           //"DI2"."SPARE1" := "BA010AZCRDI2.00";
           "DI2"."CONTROL POWER SMPS DC OK E6104PWS" := "BA010AZCRMP102.01";
           "DI2"."ET200MP I/O OUTPUT POWER TRIPPED E6154CB" := "BA010AZCRMP102.02";
           "DI2"."JUNCTION BOX CONTROL POWER TRIPPED E6180CB" := "BA010AZCRMP102.03";
           "DI2"."CLASS 2 SMPS POWER TRIPPED E6204CB" := "BA010AZCRMP102.04";
           "DI2"."CLASS 2 SMPS MONITORING E6206PWS" := "BA010AZCRMP102.05";
           "DI2"."ET200ECO PN-1 POWER TRIPPED E6220CB" := "BA010AZCRMP102.06";
           "DI2"."ET200ECO PN-2 POWER TRIPPED E6224CB" := "BA010AZCRMP102.07";
           "DI2"."ET200ECO PN-3 POWER TRIPPED E6228CB" := "BA010AZCRMP102.10";
           //"DI2"."SPARE2" := "BA010AZCRDI2.09";
           "DI2"."PANEL FAN POWER TRIPPED E6304CB" := "BA010AZCRMP102.12";
           //"DI2"."SPARE3" := "BA010AZCRDI2.11";
           "DI2"."CONTROLLER POWER SMPS DC OK E6404PWS" := "BA010AZCRMP102.14";
           "DI2"."CONTROLLER DC POWER TRIPPED E6406CB" := "BA010AZCRMP102.15";
           "DI2"."SERVO CONTROL POWER TRIPPED E6416CB" := "BA010AZCRMP102.16";
           "DI2"."MANIFOLD-1 CONTROL POWER TRIPPED E6422CB" := "BA010AZCRMP102.17";
           //"DI2"."SPARE4" := "BA010AZCRDI2.16";
           "DI2"."RFID POWER TRIPPED E6456CB" := "BA010AZCRMP102.21";
           "DI2"."QR READER POWER TRIPPED E6462CB" := "BA010AZCRMP102.22";
           "DI2"."QR READER POWER TRIPPED E6468CB" := "BA010AZCRMP102.23";
           //"DI2"."SPARE5" := "BA010AZCRDI2.20";
           //"DI2"."SPARE6" := "BA010AZCRDI2.21";
           "DI2"."CONTROLLER POWER SMPS DC OK E6704PWS" := "BA010AZCRMP102.26";
           "DI2"."CONTROLLER DC POWER TRIPPED E6706CB" := "BA010AZCRMP102.27";
           "DI2"."HANDY QR READER POWER TRIPPED E6716CB" := "BA010AZCRMP102.30";
           "DI2"."VISION CONTROLLER POWER TRIPPED E6722CB" := "BA010AZCRMP102.31";
           "DI2"."LINE LASER MODULE-1 POWER TRIPPED E6728CB" := "BA010AZCRMP102.32";
           "DI2"."LINE LASER MODULE-2 POWER TRIPPED E6734CB" := "BA010AZCRMP102.33";
           "DI2"."EPC CONTROLLER-1 POWER TRIPPED E6756CB" := "BA010AZCRMP102.34";
           "DI2"."EPC CONTROLLER-2 POWER TRIPPED E6762CB" := "BA010AZCRMP102.35";
           "DI2"."EPC CONTROLLER-3 POWER TRIPPED E6768CB" := "BA010AZCRMP102.36";
           "DI2"."DRIVE-CLIQ HUB POWER TRIPPED E6774CB" := "BA010AZCRMP102.37";


       END_REGION

       REGION DI3

           "DI3"."EQUIPMENT LED POWER TRIPPED E6780CB" := "BA010AZCRMP103.00";
           "DI3"."MOTOR POWER MC COIL POWER TRIPPED E6786CB" := "BA010AZCRMP103.01";
           "DI3"."SAFETY POWER SMPS DC OK E6804PWS" := "BA010AZCRMP103.02";
           "DI3"."SAFETY DC POWER TRIPPED E6808CB" := "BA010AZCRMP103.03";
           "DI3"."ET200SP I/O SAFETY POWER TRIPPED E6816CB" := "BA010AZCRMP103.04";
           "DI3"."JUNCTION BOX CONTROL POWER TRIPPED E6836CB" := "BA010AZCRMP103.05";
           "DI3"."ET200ECO PN-SAFETY-1 POWER TRIPPED E6856CB" := "BA010AZCRMP103.06";
           //"DI3"."SPARE1" := "BA010AZCRDI3.07";
           //"DI3"."SPARE2" := "BA010AZCRDI3.08";
           //"DI3"."SPARE3" := "BA010AZCRDI3.09";
           //"DI3"."SPARE4" := "BA010AZCRDI3.10";
           //"DI3"."SPARE5" := "BA010AZCRDI3.11";
           //"DI3"."SPARE6" := "BA010AZCRDI3.12";
           //"DI3"."SPARE7" := "BA010AZCRDI3.13";
           //"DI3"."SPARE8" := "BA010AZCRDI3.14";
           //"DI3"."SPARE9" := "BA010AZCRDI3.15";
           //"DI3"."SPARE10" := "BA010AZCRDI3.16";
           //"DI3"."SPARE11" := "BA010AZCRDI3.17";
           //"DI3"."SPARE12" := "BA010AZCRDI3.18";
           //"DI3"."SPARE13" := "BA010AZCRDI3.19";
           //"DI3"."SPARE14" := "BA010AZCRDI3.20";
           //"DI3"."SPARE15" := "BA010AZCRDI3.21";
           //"DI3"."SPARE16" := "BA010AZCRDI3.22";
           //"DI3"."SPARE17" := "BA010AZCRDI3.23";
           //"DI3"."SPARE18" := "BA010AZCRDI3.24";
           //"DI3"."SPARE19" := "BA010AZCRDI3.25";
           //"DI3"."SPARE20" := "BA010AZCRDI3.26";
           //"DI3"."SPARE21" := "BA010AZCRDI3.27";
           //"DI3"."SPARE22" := "BA010AZCRDI3.28";
           //"DI3"."SPARE23" := "BA010AZCRDI3.29";
           //"DI3"."SPARE24" := "BA010AZCRDI3.30";
           //"DI3"."SPARE25" := "BA010AZCRDI3.31";


       END_REGION

       REGION DQ1

           "DQ1"."EQUIPMENT LED LAMP RELAY ON" := "BA010AZCRMP104.00";
           //"DQ1"."SPARE1" := "BA010AZCRDQ1.01";
           //"DQ1"."SPARE2" := "BA010AZCRDQ1.02";
           "DQ1"."CLASS2 SMPS ALARM RESET" := "BA010AZCRMP104.03";
           //"DQ1"."SPARE3" := "BA010AZCRDQ1.04";
           //"DQ1"."SPARE4" := "BA010AZCRDQ1.05";
           //"DQ1"."SPARE5" := "BA010AZCRDQ1.06";
           //"DQ1"."SPARE6" := "BA010AZCRDQ1.07";
           //"DQ1"."SPARE7" := "BA010AZCRDQ1.08";
           //"DQ1"."SPARE8" := "BA010AZCRDQ1.09";
           //"DQ1"."SPARE9" := "BA010AZCRDQ1.10";
           //"DQ1"."SPARE10" := "BA010AZCRDQ1.11";
           //"DQ1"."SPARE11" := "BA010AZCRDQ1.12";
           //"DQ1"."SPARE12" := "BA010AZCRDQ1.13";
           //"DQ1"."SPARE13" := "BA010AZCRDQ1.14";
           //"DQ1"."SPARE14" := "BA010AZCRDQ1.15";
           //"DQ1"."SPARE15" := "BA010AZCRDQ1.16";
           //"DQ1"."SPARE16" := "BA010AZCRDQ1.17";
           //"DQ1"."SPARE17" := "BA010AZCRDQ1.18";
           //"DQ1"."SPARE18" := "BA010AZCRDQ1.19";
           //"DQ1"."SPARE19" := "BA010AZCRDQ1.20";
           //"DQ1"."SPARE20" := "BA010AZCRDQ1.21";
           //"DQ1"."SPARE21" := "BA010AZCRDQ1.22";
           //"DQ1"."SPARE22" := "BA010AZCRDQ1.23";
           //"DQ1"."SPARE23" := "BA010AZCRDQ1.24";
           //"DQ1"."SPARE24" := "BA010AZCRDQ1.25";
           //"DQ1"."SPARE25" := "BA010AZCRDQ1.26";
           //"DQ1"."SPARE26" := "BA010AZCRDQ1.27";
           //"DQ1"."SPARE27" := "BA010AZCRDQ1.28";
           //"DQ1"."SPARE28" := "BA010AZCRDQ1.29";
           //"DQ1"."SPARE29" := "BA010AZCRDQ1.30";
           //"DQ1"."SPARE30" := "BA010AZCRDQ1.31";


       END_REGION

       REGION FDI1

           "FDI1"."MANIFOLD-1 SOL POWER MC FEEDBACK" := "BA010AZCRMP105.00";
           "FDI1"."MANIFOLD-2 SOL POWER MC FEEDBACK" := "BA010AZCRMP105.01";
           //"FDI1"."SPARE1" := "BA010AZCRFDI1.02";
           //"FDI1"."SPARE2" := "BA010AZCRFDI1.03";
           "FDI1"."FFU POWER MC 1 FEEDBACK" := "BA010AZCRMP105.04";
           "FDI1"."FFU POWER MC 2 FEEDBACK" := "BA010AZCRMP105.05";
           //"FDI1"."SPARE3" := "BA010AZCRFDI1.06";
           //"FDI1"."SPARE4" := "BA010AZCRFDI1.07";


       END_REGION

       REGION FDQ1

           "FDQ1"."MANIFOLD-1 SOL POWER MC ON" := "BA010AZCRMP106.00";
           //"FDQ1"."SPARE1" := "BA010AZCRFDQ1.01";
           //"FDQ1"."SPARE2" := "BA010AZCRFDQ1.02";
           //"FDQ1"."SPARE3" := "BA010AZCRFDQ1.03";
           "FDQ1"."FFU POWER MC ON 1" := "BA010AZCRMP106.04";
           "FDQ1"."FFU POWER MC ON 2" := "BA010AZCRMP106.05";
           //"FDQ1"."SPARE4" := "BA010AZCRFDQ1.06";
           //"FDQ1"."SPARE5" := "BA010AZCRFDQ1.07";


       END_REGION


   END_REGION
END_FUNCTION

FUNCTION_BLOCK "CallInterfaceSignals"   // FB38, LAD
TITLE = CallInterfaceSignals
AUTHOR : SICAR
FAMILY : Diag
VERSION : 1.0
// Der Baustein dient als Aufrufschnittstelle für den Funktionsbaustein „LSicar_InterfaceSignalsBool“. Er ist als Funktionsbaustein ausgeführt, um die intern aufgerufenen FBs mittels Multiinstanzen realisieren zu können.  
// Die Funktionsbausteine und das zugehörige WinCC-Bild sind für 16 Signaldatensätze („Schnittstelle Signale 01“ … „Schnittstellen Signale 16“) mit jeweils 32 boolschen Signalen vorgesehen.  
// 
// **PLC-Datentypen**  
//  LSicar_typeInterfaceSignalsBool 
//  typeInterfaceSignalsHmi 
//  LSicar _typeInterfaceSignals 
// 
// **WinCC-Diagnosebild**  
// 
// ![Icon](_Icon/reference.PNG)
// 
// siehe ..\Library Types\LSicar_InterfaceSignalsBool.pdf  
// 
//  
// 
// **Beispielaufruf**  
// Abbildung in Kontaktplan (KOP).  D:\Software\Symbols_Icons\BMPs-JPGs-PNGs\Verschiedene\symb_user_goto_transparent.pngEin lauffähiger Programm-Aufruf hierzu ist im „SICAR-StartUp“-Projekt enthalten.  
// 
// **Aufrufschnittstelle**  
// Der Baustein wird einmalig im zyklischen Programm aufgerufen.  
// 
// **Intern verwendete „Erweiterte Anweisungen / Bausteine“**  
// ..\Library Types\LSicar_InterfaceSignalsBool.pdf
// The block serves as a calling interface of the block “InterfaceSignalsBool“. The block is designed as function block in order to implement the block calls as multi-instances.
// stored: IsIECCheckEnabled true, MemoryReserve 100, SetENOAutomatically true
   VAR
      statReadValueHmi : Bool;   // HMI: Lese Signalwert / HMI: Read value signal
      statSelectSignalsHmi : USInt := 1;   // HMI: Angewählte Interface Schnittstelle (1..16) / HMI: Selected interface signals (1..16)
      statSelectSignalsOld { ExternalAccessible := 'False'; ExternalVisible := 'False'; ExternalWritable := 'False'} : USInt;   // Altwert: Angewählte Interface Schnittstelle / Old value: Selected interface signals
      statRisEdgeReadName { ExternalAccessible := 'False'; ExternalVisible := 'False'; ExternalWritable := 'False'} : Bool;   // Steigende Flanke / Rising edge
      statPosPulseReadName : Bool;   // Positiver Impuls / Positive pulse
   END_VAR
   VAR RETAIN
      statInterfaceSignalsHmi : Array[0..70] of "typeInterfaceSignalsHmi";   // HMI: Beschreibung, Wert und Symbolischer Name / HMI: Description, value and symbolic name
   END_VAR
   VAR
      instSignalsLeft { ExternalAccessible := 'False'; ExternalVisible := 'False'; ExternalWritable := 'False'} : Array[0..70] of "LAF_InterfaceSignalsBool";   // Schnittstellen Signale Bild 1 links / interface signals screen left
      instSignalsRight { ExternalAccessible := 'False'; ExternalVisible := 'False'; ExternalWritable := 'False'} : Array[0..70] of "LAF_InterfaceSignalsBool";   // Schnittstellen Signale Bild 1 rechts / interface signals screen right
   END_VAR
   VAR_TEMP
      tempLoopCounter : DInt;   // temp. Schleifenzähler / temp. Loop Counter
   END_VAR
   VAR_TEMP   // added for the SCL form of the ladder/FBD networks
      _w1 : Bool;
   END_VAR
BEGIN

REGION Network 1: Beschreibung / BLOCK INFO HEADER
   // **Betriebsart Automatik / Hand**  
   // Der Baustein ist keiner Betriebsart / Betriebsartenbereich zugeordnet.  
   // 
   // **Alarme**  
   // Der Baustein generiert keine Alarme.  
   // 
   // #### PLC-Datentypen  
   // Verwendete PLC-Datentypen für den SPS-Programmbaustein und das zugehörige WinCC-Bild.  
   // 
   // {.pageWidth}
   // ![Image](CallInterfaceSignals/de/image1.PNG)
   //  
   //  
   // #### Bausteinaufrufe 
   // Der Baustein “LSicar_InterfaceSignalsBool“ wird in diesem FB als Multi-Instanz aufgerufen, entspr. nebenstehender beispielhafter Darstellung.  
   // 
   // {.pageWidth}
   // ![Image](CallInterfaceSignals/de/image2.PNG)
   //  
   // Um einen neuen FB aufzurufen, ziehen Sie den FB in ein neues Netzwerk, wählen Sie „Multiinstanz“ aus, vergeben Sie einen Namen und parametrieren Sie den FB-Aufruf.  
   // 
   // {.pageWidth}
   // ![Image](CallInterfaceSignals/de/image3.PNG)
   //  
   //  
   // #### Weitere Hinweise 
   // 
   // #### Updateinfo 
   // 
   // #### Weitere Dokumente 
   // 
   // ![Icon](_Icon/reference.PNG)
   // 
   // ..\Library Types\LSicar_InterfaceSignalsBool.pdf
   // SIEMENS AG / (c)Copyright 2023
   // ------------------------------------------------------------------------------
   // Title:            CallInterfaceSignals (FB38)
   // Comment/Function: The block serves as a calling interface of the block “InterfaceSignalsBool“. The block is designed as function block in order to implement the block calls as multi-instances. 
   // Library/Family:   Diag
   // Author:           SICAR
   // Tested with:      ---
   // Engineering:      TIA Portal V19
   // Restrictions:     -
   // Requirements:     ---
   // ------------------------------------------------------------------------------
   // Change log table:
   // Version  | Date       | Expert in charge       | Changes applied
   // ---------|------------|------------------------|------------------------------
   // 01.00.00 | 11.12.2023 | SICAR
   //                         First released version
END_REGION

REGION Network 2: DESCRIPTION
   // Function block and corresponding WinCC screen are prepared for 16 data sets (“InterfaceSignals01“ through .”InterfaceSignals16“) with 32 Boolean signals each.  
   // 
   // **PLC-Data types**   
   // 
   // * LSicar_typeInterfaceSignalsBool 
   // * LSicar _typeInterfaceSignals 
   // * typeInterfaceSignalsHmi 
   // 
   // **WinCC-Faceplate**  
   // 
   // <None> 
   // 
   // **WinCC Diagnostic screen**   
   // 
   // See: ..\Library Types\LSicar_InterfaceSignalsBool.pdf  
   // 
   // **Block call example** 
   // 
   // View in ladder-logic (LAD), without parameter settings.  
   // An executable program call is available in the “SICAR-Startup” project.  
   // 
   // **Calling interface**  
   // 
   // The block is be called once in the cyclic program.  
   // 
   // **Internally used „Extended instructions / blocks“**  
   // 
   // See: ..\Library Types\LSicar_InterfaceSignalsBool.pdf
END_REGION

REGION Network 3: Initialisierung Loop_1 / Initialization Loop_1
   // Vorbesetzen des Schleifenindex / Preset the loop index
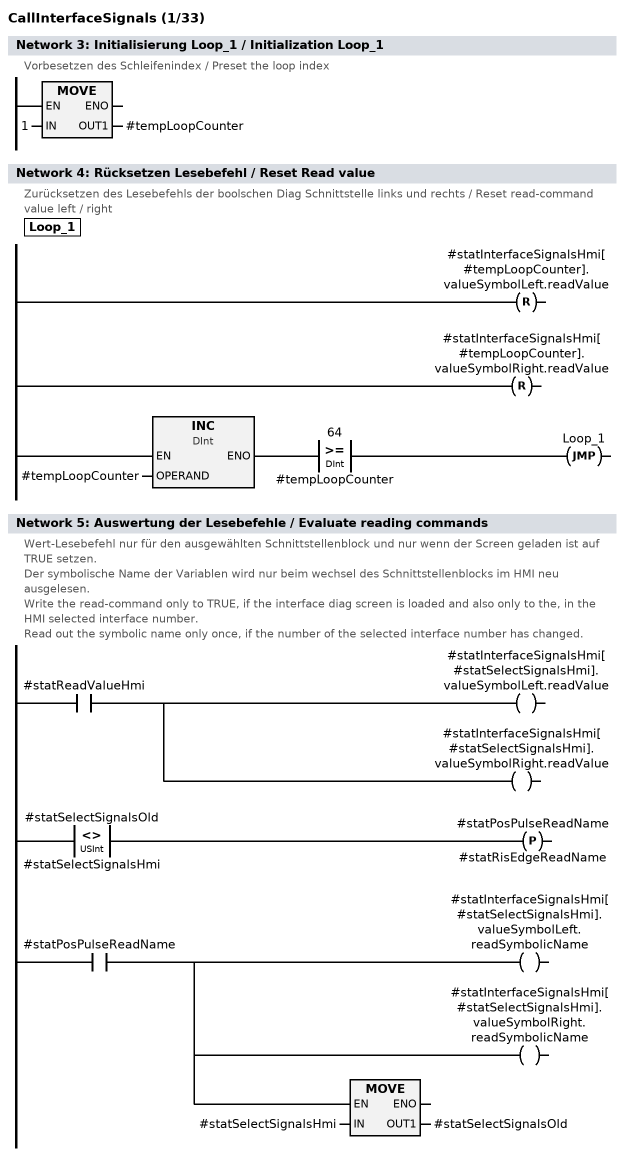
   RUNG wire#powerrail
      Move(in := 1, out1 => #tempLoopCounter)
   END_RUNG
   // the same network as SCL:
   #tempLoopCounter := 1;
END_REGION

REGION Network 4: Rücksetzen Lesebefehl / Reset Read value
   // Zurücksetzen des Lesebefehls der boolschen Diag Schnittstelle links und rechts / Reset read-command value left / right
   Label( Loop_1 )
   RUNG wire#powerrail
      R_Coil( #statInterfaceSignalsHmi[#tempLoopCounter].valueSymbolLeft.readValue )
   END_RUNG
   RUNG wire#powerrail
      R_Coil( #statInterfaceSignalsHmi[#tempLoopCounter].valueSymbolRight.readValue )
   END_RUNG
   RUNG wire#powerrail
      { S7_Templates := "DestType := DInt" } Inc( #tempLoopCounter )
      { S7_Templates := "SrcType := DInt" } GE_Contact(in1 := 64, in2 := #tempLoopCounter)
      JumpCoil( Loop_1 )
   END_RUNG
   // the same network as SCL:
   Loop_1:
   #statInterfaceSignalsHmi[#tempLoopCounter].valueSymbolLeft.readValue := FALSE;
   #statInterfaceSignalsHmi[#tempLoopCounter].valueSymbolRight.readValue := FALSE;
   #tempLoopCounter := #tempLoopCounter + 1;
   IF 64 >= #tempLoopCounter THEN GOTO Loop_1; END_IF;
END_REGION

REGION Network 5: Auswertung der Lesebefehle / Evaluate reading commands
   // Wert-Lesebefehl nur für den ausgewählten Schnittstellenblock und nur wenn der Screen geladen ist auf TRUE setzen.
   // Der symbolische Name der Variablen wird nur beim wechsel des Schnittstellenblocks im HMI neu ausgelesen.
   // Write the read-command only to TRUE, if the interface diag screen is loaded and also only to the, in the HMI selected interface number.
   // Read out the symbolic name only once, if the number of the selected interface number has changed.
   #statInterfaceSignalsHmi[#statSelectSignalsHmi].valueSymbolLeft.readValue := #statReadValueHmi;
   #statInterfaceSignalsHmi[#statSelectSignalsHmi].valueSymbolRight.readValue := #statReadValueHmi;
   #_w1 := #statSelectSignalsOld <> #statSelectSignalsHmi;
   #statPosPulseReadName := #_w1 AND NOT #statRisEdgeReadName;   // rising edge
   #statRisEdgeReadName := #_w1;
   #statInterfaceSignalsHmi[#statSelectSignalsHmi].valueSymbolLeft.readSymbolicName := #statPosPulseReadName;
   #statInterfaceSignalsHmi[#statSelectSignalsHmi].valueSymbolRight.readSymbolicName := #statPosPulseReadName;
   IF #statPosPulseReadName THEN #statSelectSignalsOld := #statSelectSignalsHmi; END_IF;
END_REGION

REGION Network 6: Interface Signals 01 -Example: Model PosDev+Lifter - IN/OUT- / Interface Signals Stack30
   // Aufruf des Schnittstellen Signal Bausteins Ba-Bereich 1 / Call the interface signals bool blocks of system tags
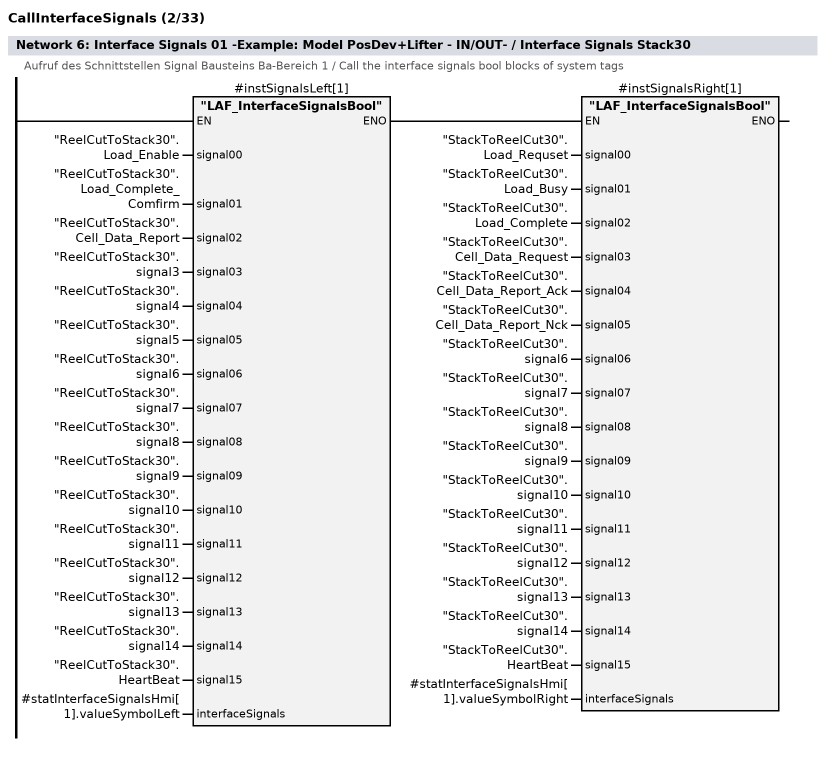
   RUNG wire#powerrail
      #instSignalsLeft[1](signal00 := "ReelCutToStack30".Load_Enable, signal01 := "ReelCutToStack30".Load_Complete_Comfirm, signal02 := "ReelCutToStack30".Cell_Data_Report, signal03 := "ReelCutToStack30".signal3, signal04 := "ReelCutToStack30".signal4, signal05 := "ReelCutToStack30".signal5, signal06 := "ReelCutToStack30".signal6, signal07 := "ReelCutToStack30".signal7, signal08 := "ReelCutToStack30".signal8, signal09 := "ReelCutToStack30".signal9, signal10 := "ReelCutToStack30".signal10, signal11 := "ReelCutToStack30".signal11, signal12 := "ReelCutToStack30".signal12, signal13 := "ReelCutToStack30".signal13, signal14 := "ReelCutToStack30".signal14, signal15 := "ReelCutToStack30".HeartBeat, interfaceSignals := #statInterfaceSignalsHmi[1].valueSymbolLeft)
      #instSignalsRight[1](signal00 := "StackToReelCut30".Load_Requset, signal01 := "StackToReelCut30".Load_Busy, signal02 := "StackToReelCut30".Load_Complete, signal03 := "StackToReelCut30".Cell_Data_Request, signal04 := "StackToReelCut30".Cell_Data_Report_Ack, signal05 := "StackToReelCut30".Cell_Data_Report_Nck, signal06 := "StackToReelCut30".signal6, signal07 := "StackToReelCut30".signal7, signal08 := "StackToReelCut30".signal8, signal09 := "StackToReelCut30".signal9, signal10 := "StackToReelCut30".signal10, signal11 := "StackToReelCut30".signal11, signal12 := "StackToReelCut30".signal12, signal13 := "StackToReelCut30".signal13, signal14 := "StackToReelCut30".signal14, signal15 := "StackToReelCut30".HeartBeat, interfaceSignals := #statInterfaceSignalsHmi[1].valueSymbolRight)
   END_RUNG
   // the same network as SCL:
   #instSignalsLeft[1](signal00 := "ReelCutToStack30".Load_Enable,   // "LAF_InterfaceSignalsBool"
                       signal01 := "ReelCutToStack30".Load_Complete_Comfirm,
                       signal02 := "ReelCutToStack30".Cell_Data_Report,
                       signal03 := "ReelCutToStack30".signal3,
                       signal04 := "ReelCutToStack30".signal4,
                       signal05 := "ReelCutToStack30".signal5,
                       signal06 := "ReelCutToStack30".signal6,
                       signal07 := "ReelCutToStack30".signal7,
                       signal08 := "ReelCutToStack30".signal8,
                       signal09 := "ReelCutToStack30".signal9,
                       signal10 := "ReelCutToStack30".signal10,
                       signal11 := "ReelCutToStack30".signal11,
                       signal12 := "ReelCutToStack30".signal12,
                       signal13 := "ReelCutToStack30".signal13,
                       signal14 := "ReelCutToStack30".signal14,
                       signal15 := "ReelCutToStack30".HeartBeat,
                       interfaceSignals := #statInterfaceSignalsHmi[1].valueSymbolLeft,
                       ENO => #_w1);
   IF #_w1 THEN
       #instSignalsRight[1](signal00 := "StackToReelCut30".Load_Requset,   // "LAF_InterfaceSignalsBool"
                            signal01 := "StackToReelCut30".Load_Busy,
                            signal02 := "StackToReelCut30".Load_Complete,
                            signal03 := "StackToReelCut30".Cell_Data_Request,
                            signal04 := "StackToReelCut30".Cell_Data_Report_Ack,
                            signal05 := "StackToReelCut30".Cell_Data_Report_Nck,
                            signal06 := "StackToReelCut30".signal6,
                            signal07 := "StackToReelCut30".signal7,
                            signal08 := "StackToReelCut30".signal8,
                            signal09 := "StackToReelCut30".signal9,
                            signal10 := "StackToReelCut30".signal10,
                            signal11 := "StackToReelCut30".signal11,
                            signal12 := "StackToReelCut30".signal12,
                            signal13 := "StackToReelCut30".signal13,
                            signal14 := "StackToReelCut30".signal14,
                            signal15 := "StackToReelCut30".HeartBeat,
                            interfaceSignals := #statInterfaceSignalsHmi[1].valueSymbolRight);
   END_IF;
END_REGION

REGION Network 7: Interface Signals 01 -Example: Model PosDev+Lifter - IN/OUT- / Interface Signals Stack40
   // Aufruf des Schnittstellen Signal Bausteins Ba-Bereich 1 / Call the interface signals bool blocks of system tags
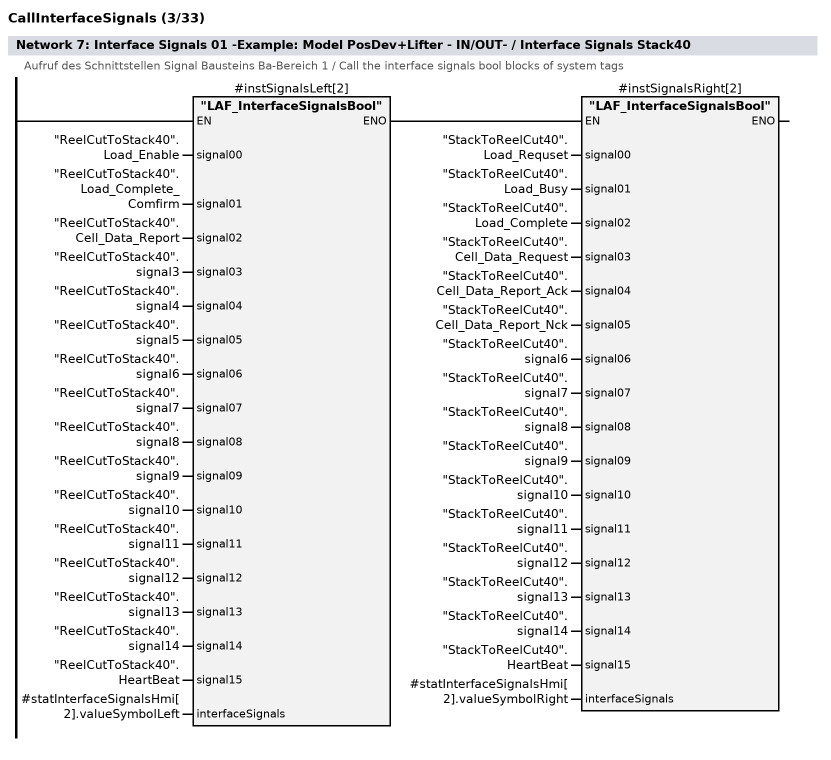
   RUNG wire#powerrail
      #instSignalsLeft[2](signal00 := "ReelCutToStack40".Load_Enable, signal01 := "ReelCutToStack40".Load_Complete_Comfirm, signal02 := "ReelCutToStack40".Cell_Data_Report, signal03 := "ReelCutToStack40".signal3, signal04 := "ReelCutToStack40".signal4, signal05 := "ReelCutToStack40".signal5, signal06 := "ReelCutToStack40".signal6, signal07 := "ReelCutToStack40".signal7, signal08 := "ReelCutToStack40".signal8, signal09 := "ReelCutToStack40".signal9, signal10 := "ReelCutToStack40".signal10, signal11 := "ReelCutToStack40".signal11, signal12 := "ReelCutToStack40".signal12, signal13 := "ReelCutToStack40".signal13, signal14 := "ReelCutToStack40".signal14, signal15 := "ReelCutToStack40".HeartBeat, interfaceSignals := #statInterfaceSignalsHmi[2].valueSymbolLeft)
      #instSignalsRight[2](signal00 := "StackToReelCut40".Load_Requset, signal01 := "StackToReelCut40".Load_Busy, signal02 := "StackToReelCut40".Load_Complete, signal03 := "StackToReelCut40".Cell_Data_Request, signal04 := "StackToReelCut40".Cell_Data_Report_Ack, signal05 := "StackToReelCut40".Cell_Data_Report_Nck, signal06 := "StackToReelCut40".signal6, signal07 := "StackToReelCut40".signal7, signal08 := "StackToReelCut40".signal8, signal09 := "StackToReelCut40".signal9, signal10 := "StackToReelCut40".signal10, signal11 := "StackToReelCut40".signal11, signal12 := "StackToReelCut40".signal12, signal13 := "StackToReelCut40".signal13, signal14 := "StackToReelCut40".signal14, signal15 := "StackToReelCut40".HeartBeat, interfaceSignals := #statInterfaceSignalsHmi[2].valueSymbolRight)
   END_RUNG
   // the same network as SCL:
   #instSignalsLeft[2](signal00 := "ReelCutToStack40".Load_Enable,   // "LAF_InterfaceSignalsBool"
                       signal01 := "ReelCutToStack40".Load_Complete_Comfirm,
                       signal02 := "ReelCutToStack40".Cell_Data_Report,
                       signal03 := "ReelCutToStack40".signal3,
                       signal04 := "ReelCutToStack40".signal4,
                       signal05 := "ReelCutToStack40".signal5,
                       signal06 := "ReelCutToStack40".signal6,
                       signal07 := "ReelCutToStack40".signal7,
                       signal08 := "ReelCutToStack40".signal8,
                       signal09 := "ReelCutToStack40".signal9,
                       signal10 := "ReelCutToStack40".signal10,
                       signal11 := "ReelCutToStack40".signal11,
                       signal12 := "ReelCutToStack40".signal12,
                       signal13 := "ReelCutToStack40".signal13,
                       signal14 := "ReelCutToStack40".signal14,
                       signal15 := "ReelCutToStack40".HeartBeat,
                       interfaceSignals := #statInterfaceSignalsHmi[2].valueSymbolLeft,
                       ENO => #_w1);
   IF #_w1 THEN
       #instSignalsRight[2](signal00 := "StackToReelCut40".Load_Requset,   // "LAF_InterfaceSignalsBool"
                            signal01 := "StackToReelCut40".Load_Busy,
                            signal02 := "StackToReelCut40".Load_Complete,
                            signal03 := "StackToReelCut40".Cell_Data_Request,
                            signal04 := "StackToReelCut40".Cell_Data_Report_Ack,
                            signal05 := "StackToReelCut40".Cell_Data_Report_Nck,
                            signal06 := "StackToReelCut40".signal6,
                            signal07 := "StackToReelCut40".signal7,
                            signal08 := "StackToReelCut40".signal8,
                            signal09 := "StackToReelCut40".signal9,
                            signal10 := "StackToReelCut40".signal10,
                            signal11 := "StackToReelCut40".signal11,
                            signal12 := "StackToReelCut40".signal12,
                            signal13 := "StackToReelCut40".signal13,
                            signal14 := "StackToReelCut40".signal14,
                            signal15 := "StackToReelCut40".HeartBeat,
                            interfaceSignals := #statInterfaceSignalsHmi[2].valueSymbolRight);
   END_IF;
END_REGION

REGION Network 8: Interface Signals 01 -Example: Rack-ET200SP Standard IN/OUT- / Interface Signals Bk01
   // Aufruf des Schnittstellen Signal Bausteins Ba-Bereich 1 / Call the interface signals bool blocks of system tags
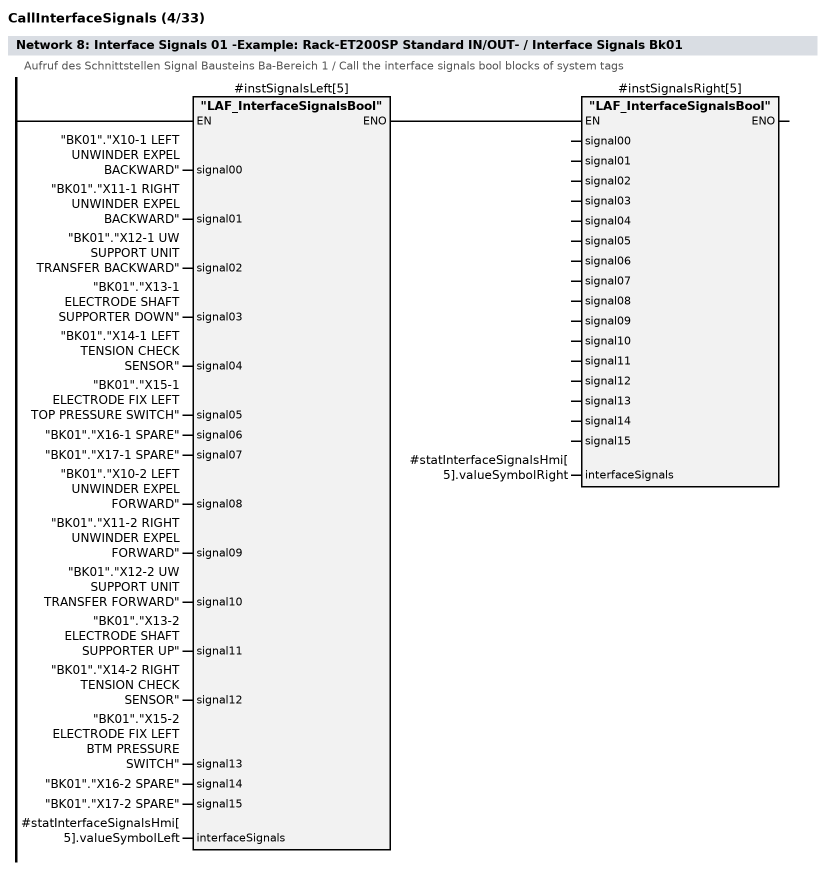
   RUNG wire#powerrail
      #instSignalsLeft[5](signal00 := "BK01"."X10-1 LEFT UNWINDER EXPEL BACKWARD", signal01 := "BK01"."X11-1 RIGHT UNWINDER EXPEL BACKWARD", signal02 := "BK01"."X12-1 UW SUPPORT UNIT TRANSFER BACKWARD", signal03 := "BK01"."X13-1 ELECTRODE SHAFT SUPPORTER DOWN", signal04 := "BK01"."X14-1 LEFT TENSION CHECK SENSOR", signal05 := "BK01"."X15-1 ELECTRODE FIX LEFT TOP PRESSURE SWITCH", signal06 := "BK01"."X16-1 SPARE", signal07 := "BK01"."X17-1 SPARE", signal08 := "BK01"."X10-2 LEFT UNWINDER EXPEL FORWARD", signal09 := "BK01"."X11-2 RIGHT UNWINDER EXPEL FORWARD", signal10 := "BK01"."X12-2 UW SUPPORT UNIT TRANSFER FORWARD", signal11 := "BK01"."X13-2 ELECTRODE SHAFT SUPPORTER UP", signal12 := "BK01"."X14-2 RIGHT TENSION CHECK SENSOR", signal13 := "BK01"."X15-2 ELECTRODE FIX LEFT BTM PRESSURE SWITCH", signal14 := "BK01"."X16-2 SPARE", signal15 := "BK01"."X17-2 SPARE", interfaceSignals := #statInterfaceSignalsHmi[5].valueSymbolLeft)
      #instSignalsRight[5](signal00 :=, signal01 :=, signal02 :=, signal03 :=, signal04 :=, signal05 :=, signal06 :=, signal07 :=, signal08 :=, signal09 :=, signal10 :=, signal11 :=, signal12 :=, signal13 :=, signal14 :=, signal15 :=, interfaceSignals := #statInterfaceSignalsHmi[5].valueSymbolRight)
   END_RUNG
   // the same network as SCL:
   #instSignalsLeft[5](signal00 := "BK01"."X10-1 LEFT UNWINDER EXPEL BACKWARD",   // "LAF_InterfaceSignalsBool"
                       signal01 := "BK01"."X11-1 RIGHT UNWINDER EXPEL BACKWARD",
                       signal02 := "BK01"."X12-1 UW SUPPORT UNIT TRANSFER BACKWARD",
                       signal03 := "BK01"."X13-1 ELECTRODE SHAFT SUPPORTER DOWN",
                       signal04 := "BK01"."X14-1 LEFT TENSION CHECK SENSOR",
                       signal05 := "BK01"."X15-1 ELECTRODE FIX LEFT TOP PRESSURE SWITCH",
                       signal06 := "BK01"."X16-1 SPARE",
                       signal07 := "BK01"."X17-1 SPARE",
                       signal08 := "BK01"."X10-2 LEFT UNWINDER EXPEL FORWARD",
                       signal09 := "BK01"."X11-2 RIGHT UNWINDER EXPEL FORWARD",
                       signal10 := "BK01"."X12-2 UW SUPPORT UNIT TRANSFER FORWARD",
                       signal11 := "BK01"."X13-2 ELECTRODE SHAFT SUPPORTER UP",
                       signal12 := "BK01"."X14-2 RIGHT TENSION CHECK SENSOR",
                       signal13 := "BK01"."X15-2 ELECTRODE FIX LEFT BTM PRESSURE SWITCH",
                       signal14 := "BK01"."X16-2 SPARE",
                       signal15 := "BK01"."X17-2 SPARE",
                       interfaceSignals := #statInterfaceSignalsHmi[5].valueSymbolLeft,
                       ENO => #_w1);
   IF #_w1 THEN
       #instSignalsRight[5](interfaceSignals := #statInterfaceSignalsHmi[5].valueSymbolRight);   // "LAF_InterfaceSignalsBool"
   END_IF;
END_REGION

REGION Network 9: Interface Signals Bk02
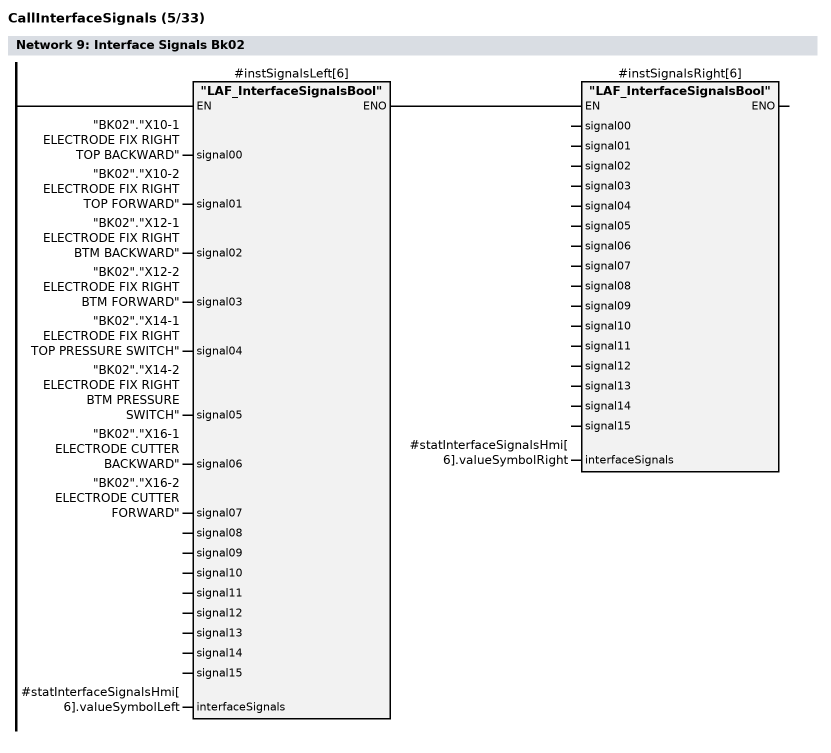
   RUNG wire#powerrail
      #instSignalsLeft[6](signal00 := "BK02"."X10-1 ELECTRODE FIX RIGHT TOP BACKWARD", signal01 := "BK02"."X10-2 ELECTRODE FIX RIGHT TOP FORWARD", signal02 := "BK02"."X12-1 ELECTRODE FIX RIGHT BTM BACKWARD", signal03 := "BK02"."X12-2 ELECTRODE FIX RIGHT BTM FORWARD", signal04 := "BK02"."X14-1 ELECTRODE FIX RIGHT TOP PRESSURE SWITCH", signal05 := "BK02"."X14-2 ELECTRODE FIX RIGHT BTM PRESSURE SWITCH", signal06 := "BK02"."X16-1 ELECTRODE CUTTER BACKWARD", signal07 := "BK02"."X16-2 ELECTRODE CUTTER FORWARD", signal08 :=, signal09 :=, signal10 :=, signal11 :=, signal12 :=, signal13 :=, signal14 :=, signal15 :=, interfaceSignals := #statInterfaceSignalsHmi[6].valueSymbolLeft)
      #instSignalsRight[6](signal00 :=, signal01 :=, signal02 :=, signal03 :=, signal04 :=, signal05 :=, signal06 :=, signal07 :=, signal08 :=, signal09 :=, signal10 :=, signal11 :=, signal12 :=, signal13 :=, signal14 :=, signal15 :=, interfaceSignals := #statInterfaceSignalsHmi[6].valueSymbolRight)
   END_RUNG
   // the same network as SCL:
   #instSignalsLeft[6](signal00 := "BK02"."X10-1 ELECTRODE FIX RIGHT TOP BACKWARD",   // "LAF_InterfaceSignalsBool"
                       signal01 := "BK02"."X10-2 ELECTRODE FIX RIGHT TOP FORWARD",
                       signal02 := "BK02"."X12-1 ELECTRODE FIX RIGHT BTM BACKWARD",
                       signal03 := "BK02"."X12-2 ELECTRODE FIX RIGHT BTM FORWARD",
                       signal04 := "BK02"."X14-1 ELECTRODE FIX RIGHT TOP PRESSURE SWITCH",
                       signal05 := "BK02"."X14-2 ELECTRODE FIX RIGHT BTM PRESSURE SWITCH",
                       signal06 := "BK02"."X16-1 ELECTRODE CUTTER BACKWARD",
                       signal07 := "BK02"."X16-2 ELECTRODE CUTTER FORWARD",
                       interfaceSignals := #statInterfaceSignalsHmi[6].valueSymbolLeft,
                       ENO => #_w1);
   IF #_w1 THEN
       #instSignalsRight[6](interfaceSignals := #statInterfaceSignalsHmi[6].valueSymbolRight);   // "LAF_InterfaceSignalsBool"
   END_IF;
END_REGION

REGION Network 10: Interface Signals 03 -Example: System flags & Clock flags- / Interface Signals Bk03
   // Aufruf des Schnittstellen Signal Bausteins für die Systemvariablen / Call the interface signals bool blocks of system tags
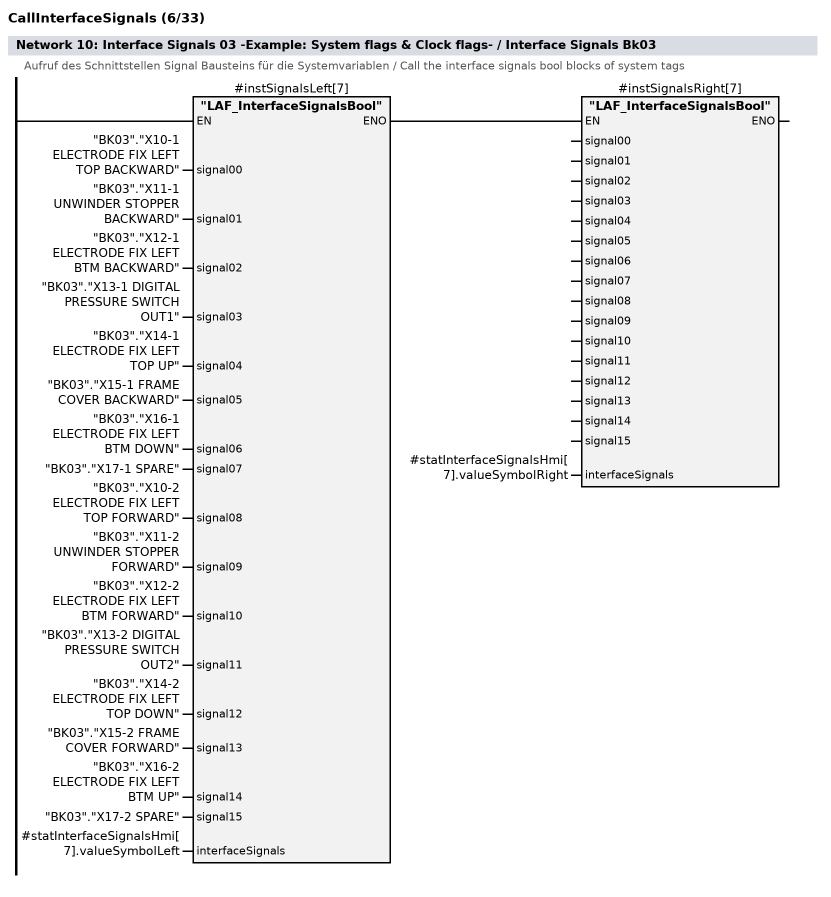
   RUNG wire#powerrail
      #instSignalsLeft[7](signal00 := "BK03"."X10-1 ELECTRODE FIX LEFT TOP BACKWARD", signal01 := "BK03"."X11-1 UNWINDER STOPPER BACKWARD", signal02 := "BK03"."X12-1 ELECTRODE FIX LEFT BTM BACKWARD", signal03 := "BK03"."X13-1 DIGITAL PRESSURE SWITCH OUT1", signal04 := "BK03"."X14-1 ELECTRODE FIX LEFT TOP UP", signal05 := "BK03"."X15-1 FRAME COVER BACKWARD", signal06 := "BK03"."X16-1 ELECTRODE FIX LEFT BTM DOWN", signal07 := "BK03"."X17-1 SPARE", signal08 := "BK03"."X10-2 ELECTRODE FIX LEFT TOP FORWARD", signal09 := "BK03"."X11-2 UNWINDER STOPPER FORWARD", signal10 := "BK03"."X12-2 ELECTRODE FIX LEFT BTM FORWARD", signal11 := "BK03"."X13-2 DIGITAL PRESSURE SWITCH OUT2", signal12 := "BK03"."X14-2 ELECTRODE FIX LEFT TOP DOWN", signal13 := "BK03"."X15-2 FRAME COVER FORWARD", signal14 := "BK03"."X16-2 ELECTRODE FIX LEFT BTM UP", signal15 := "BK03"."X17-2 SPARE", interfaceSignals := #statInterfaceSignalsHmi[7].valueSymbolLeft)
      #instSignalsRight[7](signal00 :=, signal01 :=, signal02 :=, signal03 :=, signal04 :=, signal05 :=, signal06 :=, signal07 :=, signal08 :=, signal09 :=, signal10 :=, signal11 :=, signal12 :=, signal13 :=, signal14 :=, signal15 :=, interfaceSignals := #statInterfaceSignalsHmi[7].valueSymbolRight)
   END_RUNG
   // the same network as SCL:
   #instSignalsLeft[7](signal00 := "BK03"."X10-1 ELECTRODE FIX LEFT TOP BACKWARD",   // "LAF_InterfaceSignalsBool"
                       signal01 := "BK03"."X11-1 UNWINDER STOPPER BACKWARD",
                       signal02 := "BK03"."X12-1 ELECTRODE FIX LEFT BTM BACKWARD",
                       signal03 := "BK03"."X13-1 DIGITAL PRESSURE SWITCH OUT1",
                       signal04 := "BK03"."X14-1 ELECTRODE FIX LEFT TOP UP",
                       signal05 := "BK03"."X15-1 FRAME COVER BACKWARD",
                       signal06 := "BK03"."X16-1 ELECTRODE FIX LEFT BTM DOWN",
                       signal07 := "BK03"."X17-1 SPARE",
                       signal08 := "BK03"."X10-2 ELECTRODE FIX LEFT TOP FORWARD",
                       signal09 := "BK03"."X11-2 UNWINDER STOPPER FORWARD",
                       signal10 := "BK03"."X12-2 ELECTRODE FIX LEFT BTM FORWARD",
                       signal11 := "BK03"."X13-2 DIGITAL PRESSURE SWITCH OUT2",
                       signal12 := "BK03"."X14-2 ELECTRODE FIX LEFT TOP DOWN",
                       signal13 := "BK03"."X15-2 FRAME COVER FORWARD",
                       signal14 := "BK03"."X16-2 ELECTRODE FIX LEFT BTM UP",
                       signal15 := "BK03"."X17-2 SPARE",
                       interfaceSignals := #statInterfaceSignalsHmi[7].valueSymbolLeft,
                       ENO => #_w1);
   IF #_w1 THEN
       #instSignalsRight[7](interfaceSignals := #statInterfaceSignalsHmi[7].valueSymbolRight);   // "LAF_InterfaceSignalsBool"
   END_IF;
END_REGION

REGION Network 11: Interface Signals 03 -Example: System flags & Clock flags- / Interface Signals Bk04
   // Aufruf des Schnittstellen Signal Bausteins für die Systemvariablen / Call the interface signals bool blocks of system tags
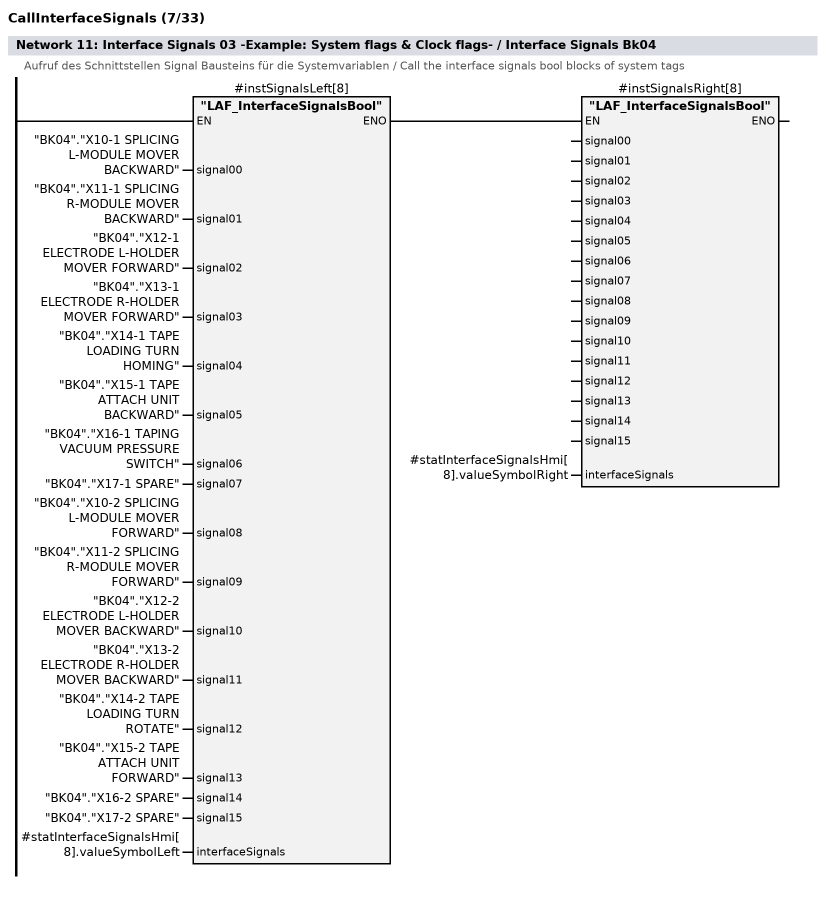
   RUNG wire#powerrail
      #instSignalsLeft[8](signal00 := "BK04"."X10-1 SPLICING L-MODULE MOVER BACKWARD", signal01 := "BK04"."X11-1 SPLICING R-MODULE MOVER BACKWARD", signal02 := "BK04"."X12-1 ELECTRODE L-HOLDER MOVER FORWARD", signal03 := "BK04"."X13-1 ELECTRODE R-HOLDER MOVER FORWARD", signal04 := "BK04"."X14-1 TAPE LOADING TURN HOMING", signal05 := "BK04"."X15-1 TAPE ATTACH UNIT BACKWARD", signal06 := "BK04"."X16-1 TAPING VACUUM PRESSURE SWITCH", signal07 := "BK04"."X17-1 SPARE", signal08 := "BK04"."X10-2 SPLICING L-MODULE MOVER FORWARD", signal09 := "BK04"."X11-2 SPLICING R-MODULE MOVER FORWARD", signal10 := "BK04"."X12-2 ELECTRODE L-HOLDER MOVER BACKWARD", signal11 := "BK04"."X13-2 ELECTRODE R-HOLDER MOVER BACKWARD", signal12 := "BK04"."X14-2 TAPE LOADING TURN ROTATE", signal13 := "BK04"."X15-2 TAPE ATTACH UNIT FORWARD", signal14 := "BK04"."X16-2 SPARE", signal15 := "BK04"."X17-2 SPARE", interfaceSignals := #statInterfaceSignalsHmi[8].valueSymbolLeft)
      #instSignalsRight[8](signal00 :=, signal01 :=, signal02 :=, signal03 :=, signal04 :=, signal05 :=, signal06 :=, signal07 :=, signal08 :=, signal09 :=, signal10 :=, signal11 :=, signal12 :=, signal13 :=, signal14 :=, signal15 :=, interfaceSignals := #statInterfaceSignalsHmi[8].valueSymbolRight)
   END_RUNG
   // the same network as SCL:
   #instSignalsLeft[8](signal00 := "BK04"."X10-1 SPLICING L-MODULE MOVER BACKWARD",   // "LAF_InterfaceSignalsBool"
                       signal01 := "BK04"."X11-1 SPLICING R-MODULE MOVER BACKWARD",
                       signal02 := "BK04"."X12-1 ELECTRODE L-HOLDER MOVER FORWARD",
                       signal03 := "BK04"."X13-1 ELECTRODE R-HOLDER MOVER FORWARD",
                       signal04 := "BK04"."X14-1 TAPE LOADING TURN HOMING",
                       signal05 := "BK04"."X15-1 TAPE ATTACH UNIT BACKWARD",
                       signal06 := "BK04"."X16-1 TAPING VACUUM PRESSURE SWITCH",
                       signal07 := "BK04"."X17-1 SPARE",
                       signal08 := "BK04"."X10-2 SPLICING L-MODULE MOVER FORWARD",
                       signal09 := "BK04"."X11-2 SPLICING R-MODULE MOVER FORWARD",
                       signal10 := "BK04"."X12-2 ELECTRODE L-HOLDER MOVER BACKWARD",
                       signal11 := "BK04"."X13-2 ELECTRODE R-HOLDER MOVER BACKWARD",
                       signal12 := "BK04"."X14-2 TAPE LOADING TURN ROTATE",
                       signal13 := "BK04"."X15-2 TAPE ATTACH UNIT FORWARD",
                       signal14 := "BK04"."X16-2 SPARE",
                       signal15 := "BK04"."X17-2 SPARE",
                       interfaceSignals := #statInterfaceSignalsHmi[8].valueSymbolLeft,
                       ENO => #_w1);
   IF #_w1 THEN
       #instSignalsRight[8](interfaceSignals := #statInterfaceSignalsHmi[8].valueSymbolRight);   // "LAF_InterfaceSignalsBool"
   END_IF;
END_REGION

REGION Network 12: Interface Signals 04 -Example: Model Flex-Pro-Line - IN/OUT- / Interface Signals Bk05
   // Aufruf des Schnittstellen Signal Bausteins Ba-Bereich 4 / Call the interface signals bool blocks of opmode 4
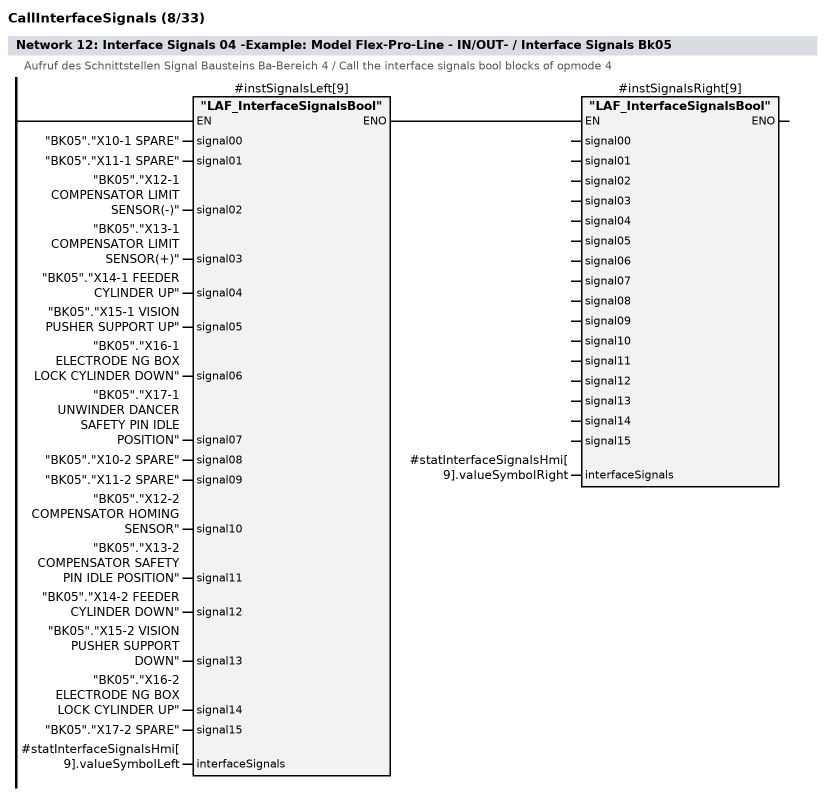
   RUNG wire#powerrail
      #instSignalsLeft[9](signal00 := "BK05"."X10-1 SPARE", signal01 := "BK05"."X11-1 SPARE", signal02 := "BK05"."X12-1 COMPENSATOR LIMIT SENSOR(-)", signal03 := "BK05"."X13-1 COMPENSATOR LIMIT SENSOR(+)", signal04 := "BK05"."X14-1 FEEDER CYLINDER UP", signal05 := "BK05"."X15-1 VISION PUSHER SUPPORT UP", signal06 := "BK05"."X16-1 ELECTRODE NG BOX LOCK CYLINDER DOWN", signal07 := "BK05"."X17-1 UNWINDER DANCER SAFETY PIN IDLE POSITION", signal08 := "BK05"."X10-2 SPARE", signal09 := "BK05"."X11-2 SPARE", signal10 := "BK05"."X12-2 COMPENSATOR HOMING SENSOR", signal11 := "BK05"."X13-2 COMPENSATOR SAFETY PIN IDLE POSITION", signal12 := "BK05"."X14-2 FEEDER CYLINDER DOWN", signal13 := "BK05"."X15-2 VISION PUSHER SUPPORT DOWN", signal14 := "BK05"."X16-2 ELECTRODE NG BOX LOCK CYLINDER UP", signal15 := "BK05"."X17-2 SPARE", interfaceSignals := #statInterfaceSignalsHmi[9].valueSymbolLeft)
      #instSignalsRight[9](signal00 :=, signal01 :=, signal02 :=, signal03 :=, signal04 :=, signal05 :=, signal06 :=, signal07 :=, signal08 :=, signal09 :=, signal10 :=, signal11 :=, signal12 :=, signal13 :=, signal14 :=, signal15 :=, interfaceSignals := #statInterfaceSignalsHmi[9].valueSymbolRight)
   END_RUNG
   // the same network as SCL:
   #instSignalsLeft[9](signal00 := "BK05"."X10-1 SPARE",   // "LAF_InterfaceSignalsBool"
                       signal01 := "BK05"."X11-1 SPARE",
                       signal02 := "BK05"."X12-1 COMPENSATOR LIMIT SENSOR(-)",
                       signal03 := "BK05"."X13-1 COMPENSATOR LIMIT SENSOR(+)",
                       signal04 := "BK05"."X14-1 FEEDER CYLINDER UP",
                       signal05 := "BK05"."X15-1 VISION PUSHER SUPPORT UP",
                       signal06 := "BK05"."X16-1 ELECTRODE NG BOX LOCK CYLINDER DOWN",
                       signal07 := "BK05"."X17-1 UNWINDER DANCER SAFETY PIN IDLE POSITION",
                       signal08 := "BK05"."X10-2 SPARE",
                       signal09 := "BK05"."X11-2 SPARE",
                       signal10 := "BK05"."X12-2 COMPENSATOR HOMING SENSOR",
                       signal11 := "BK05"."X13-2 COMPENSATOR SAFETY PIN IDLE POSITION",
                       signal12 := "BK05"."X14-2 FEEDER CYLINDER DOWN",
                       signal13 := "BK05"."X15-2 VISION PUSHER SUPPORT DOWN",
                       signal14 := "BK05"."X16-2 ELECTRODE NG BOX LOCK CYLINDER UP",
                       signal15 := "BK05"."X17-2 SPARE",
                       interfaceSignals := #statInterfaceSignalsHmi[9].valueSymbolLeft,
                       ENO => #_w1);
   IF #_w1 THEN
       #instSignalsRight[9](interfaceSignals := #statInterfaceSignalsHmi[9].valueSymbolRight);   // "LAF_InterfaceSignalsBool"
   END_IF;
END_REGION

REGION Network 13: Interface Signals 04 -Example: Model Flex-Pro-Line - IN/OUT- / Interface Signals Bk06
   // Aufruf des Schnittstellen Signal Bausteins Ba-Bereich 4 / Call the interface signals bool blocks of opmode 4
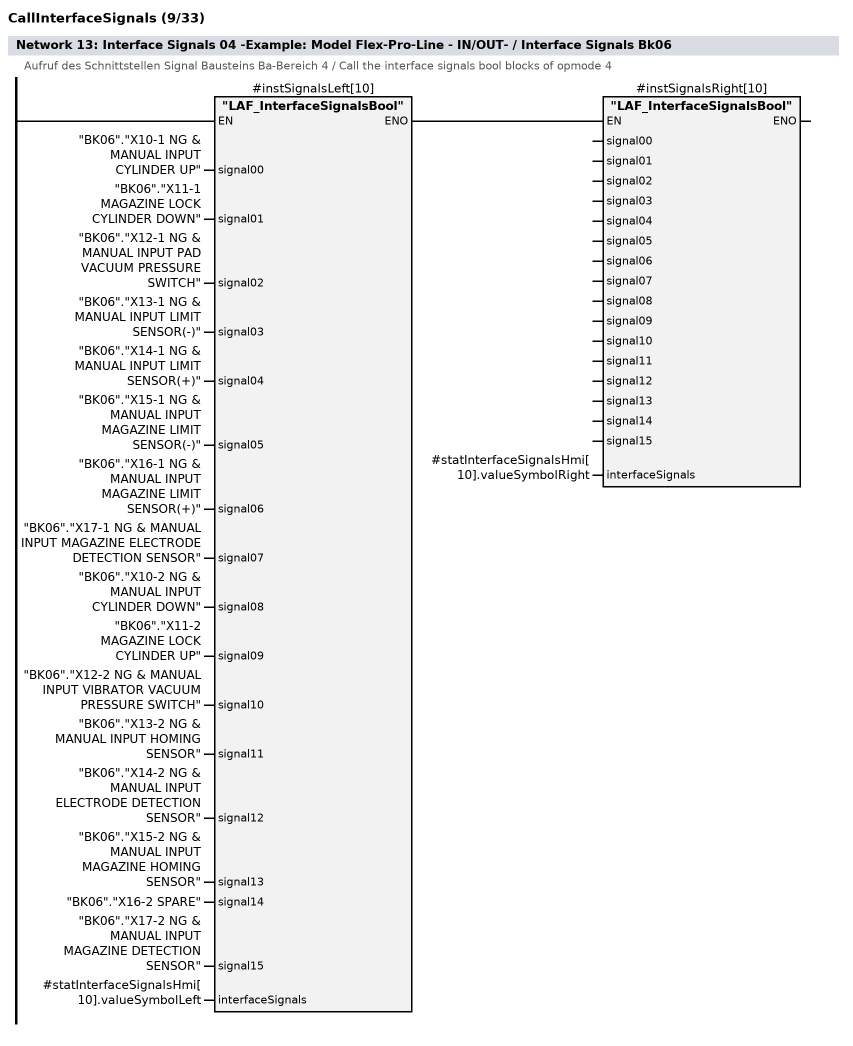
   RUNG wire#powerrail
      #instSignalsLeft[10](signal00 := "BK06"."X10-1 NG & MANUAL INPUT CYLINDER UP", signal01 := "BK06"."X11-1 MAGAZINE LOCK CYLINDER DOWN", signal02 := "BK06"."X12-1 NG & MANUAL INPUT PAD VACUUM PRESSURE SWITCH", signal03 := "BK06"."X13-1 NG & MANUAL INPUT LIMIT SENSOR(-)", signal04 := "BK06"."X14-1 NG & MANUAL INPUT LIMIT SENSOR(+)", signal05 := "BK06"."X15-1 NG & MANUAL INPUT MAGAZINE LIMIT SENSOR(-)", signal06 := "BK06"."X16-1 NG & MANUAL INPUT MAGAZINE LIMIT SENSOR(+)", signal07 := "BK06"."X17-1 NG & MANUAL INPUT MAGAZINE ELECTRODE DETECTION SENSOR", signal08 := "BK06"."X10-2 NG & MANUAL INPUT CYLINDER DOWN", signal09 := "BK06"."X11-2 MAGAZINE LOCK CYLINDER UP", signal10 := "BK06"."X12-2 NG & MANUAL INPUT VIBRATOR VACUUM PRESSURE SWITCH", signal11 := "BK06"."X13-2 NG & MANUAL INPUT HOMING SENSOR", signal12 := "BK06"."X14-2 NG & MANUAL INPUT ELECTRODE DETECTION SENSOR", signal13 := "BK06"."X15-2 NG & MANUAL INPUT MAGAZINE HOMING SENSOR", signal14 := "BK06"."X16-2 SPARE", signal15 := "BK06"."X17-2 NG & MANUAL INPUT MAGAZINE DETECTION SENSOR", interfaceSignals := #statInterfaceSignalsHmi[10].valueSymbolLeft)
      #instSignalsRight[10](signal00 :=, signal01 :=, signal02 :=, signal03 :=, signal04 :=, signal05 :=, signal06 :=, signal07 :=, signal08 :=, signal09 :=, signal10 :=, signal11 :=, signal12 :=, signal13 :=, signal14 :=, signal15 :=, interfaceSignals := #statInterfaceSignalsHmi[10].valueSymbolRight)
   END_RUNG
   // the same network as SCL:
   #instSignalsLeft[10](signal00 := "BK06"."X10-1 NG & MANUAL INPUT CYLINDER UP",   // "LAF_InterfaceSignalsBool"
                        signal01 := "BK06"."X11-1 MAGAZINE LOCK CYLINDER DOWN",
                        signal02 := "BK06"."X12-1 NG & MANUAL INPUT PAD VACUUM PRESSURE SWITCH",
                        signal03 := "BK06"."X13-1 NG & MANUAL INPUT LIMIT SENSOR(-)",
                        signal04 := "BK06"."X14-1 NG & MANUAL INPUT LIMIT SENSOR(+)",
                        signal05 := "BK06"."X15-1 NG & MANUAL INPUT MAGAZINE LIMIT SENSOR(-)",
                        signal06 := "BK06"."X16-1 NG & MANUAL INPUT MAGAZINE LIMIT SENSOR(+)",
                        signal07 := "BK06"."X17-1 NG & MANUAL INPUT MAGAZINE ELECTRODE DETECTION SENSOR",
                        signal08 := "BK06"."X10-2 NG & MANUAL INPUT CYLINDER DOWN",
                        signal09 := "BK06"."X11-2 MAGAZINE LOCK CYLINDER UP",
                        signal10 := "BK06"."X12-2 NG & MANUAL INPUT VIBRATOR VACUUM PRESSURE SWITCH",
                        signal11 := "BK06"."X13-2 NG & MANUAL INPUT HOMING SENSOR",
                        signal12 := "BK06"."X14-2 NG & MANUAL INPUT ELECTRODE DETECTION SENSOR",
                        signal13 := "BK06"."X15-2 NG & MANUAL INPUT MAGAZINE HOMING SENSOR",
                        signal14 := "BK06"."X16-2 SPARE",
                        signal15 := "BK06"."X17-2 NG & MANUAL INPUT MAGAZINE DETECTION SENSOR",
                        interfaceSignals := #statInterfaceSignalsHmi[10].valueSymbolLeft,
                        ENO => #_w1);
   IF #_w1 THEN
       #instSignalsRight[10](interfaceSignals := #statInterfaceSignalsHmi[10].valueSymbolRight);   // "LAF_InterfaceSignalsBool"
   END_IF;
END_REGION

REGION Network 14: Interface Signals 05 -Example: Model Flex-Pro-Line - IN/OUT- / Interface Signals Bk07
   // Aufruf des Schnittstellen Signal Bausteins Ba-Bereich 4 / Call the interface signals bool blocks of opmode 5
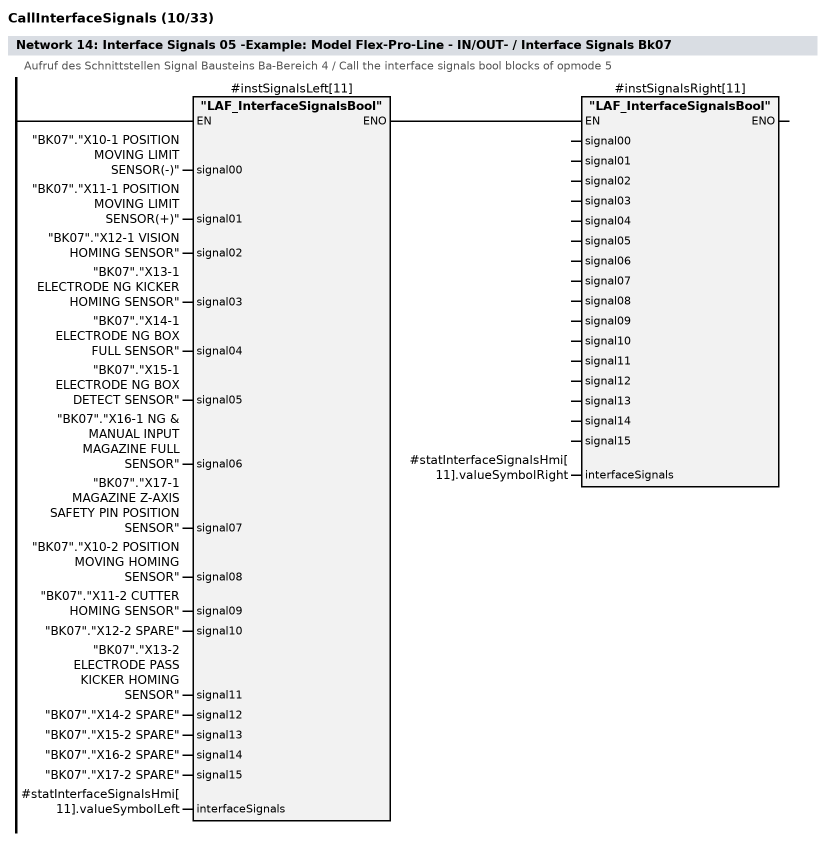
   RUNG wire#powerrail
      #instSignalsLeft[11](signal00 := "BK07"."X10-1 POSITION MOVING LIMIT SENSOR(-)", signal01 := "BK07"."X11-1 POSITION MOVING LIMIT SENSOR(+)", signal02 := "BK07"."X12-1 VISION HOMING SENSOR", signal03 := "BK07"."X13-1 ELECTRODE NG KICKER HOMING SENSOR", signal04 := "BK07"."X14-1 ELECTRODE NG BOX FULL SENSOR", signal05 := "BK07"."X15-1 ELECTRODE NG BOX DETECT SENSOR", signal06 := "BK07"."X16-1 NG & MANUAL INPUT MAGAZINE FULL SENSOR", signal07 := "BK07"."X17-1 MAGAZINE Z-AXIS SAFETY PIN POSITION SENSOR", signal08 := "BK07"."X10-2 POSITION MOVING HOMING SENSOR", signal09 := "BK07"."X11-2 CUTTER HOMING SENSOR", signal10 := "BK07"."X12-2 SPARE", signal11 := "BK07"."X13-2 ELECTRODE PASS KICKER HOMING SENSOR", signal12 := "BK07"."X14-2 SPARE", signal13 := "BK07"."X15-2 SPARE", signal14 := "BK07"."X16-2 SPARE", signal15 := "BK07"."X17-2 SPARE", interfaceSignals := #statInterfaceSignalsHmi[11].valueSymbolLeft)
      #instSignalsRight[11](signal00 :=, signal01 :=, signal02 :=, signal03 :=, signal04 :=, signal05 :=, signal06 :=, signal07 :=, signal08 :=, signal09 :=, signal10 :=, signal11 :=, signal12 :=, signal13 :=, signal14 :=, signal15 :=, interfaceSignals := #statInterfaceSignalsHmi[11].valueSymbolRight)
   END_RUNG
   // the same network as SCL:
   #instSignalsLeft[11](signal00 := "BK07"."X10-1 POSITION MOVING LIMIT SENSOR(-)",   // "LAF_InterfaceSignalsBool"
                        signal01 := "BK07"."X11-1 POSITION MOVING LIMIT SENSOR(+)",
                        signal02 := "BK07"."X12-1 VISION HOMING SENSOR",
                        signal03 := "BK07"."X13-1 ELECTRODE NG KICKER HOMING SENSOR",
                        signal04 := "BK07"."X14-1 ELECTRODE NG BOX FULL SENSOR",
                        signal05 := "BK07"."X15-1 ELECTRODE NG BOX DETECT SENSOR",
                        signal06 := "BK07"."X16-1 NG & MANUAL INPUT MAGAZINE FULL SENSOR",
                        signal07 := "BK07"."X17-1 MAGAZINE Z-AXIS SAFETY PIN POSITION SENSOR",
                        signal08 := "BK07"."X10-2 POSITION MOVING HOMING SENSOR",
                        signal09 := "BK07"."X11-2 CUTTER HOMING SENSOR",
                        signal10 := "BK07"."X12-2 SPARE",
                        signal11 := "BK07"."X13-2 ELECTRODE PASS KICKER HOMING SENSOR",
                        signal12 := "BK07"."X14-2 SPARE",
                        signal13 := "BK07"."X15-2 SPARE",
                        signal14 := "BK07"."X16-2 SPARE",
                        signal15 := "BK07"."X17-2 SPARE",
                        interfaceSignals := #statInterfaceSignalsHmi[11].valueSymbolLeft,
                        ENO => #_w1);
   IF #_w1 THEN
       #instSignalsRight[11](interfaceSignals := #statInterfaceSignalsHmi[11].valueSymbolRight);   // "LAF_InterfaceSignalsBool"
   END_IF;
END_REGION

REGION Network 15: Interface Signals 05 -Example: Model Flex-Pro-Line - IN/OUT- / Interface Signals Bk08
   // Aufruf des Schnittstellen Signal Bausteins Ba-Bereich 4 / Call the interface signals bool blocks of opmode 9
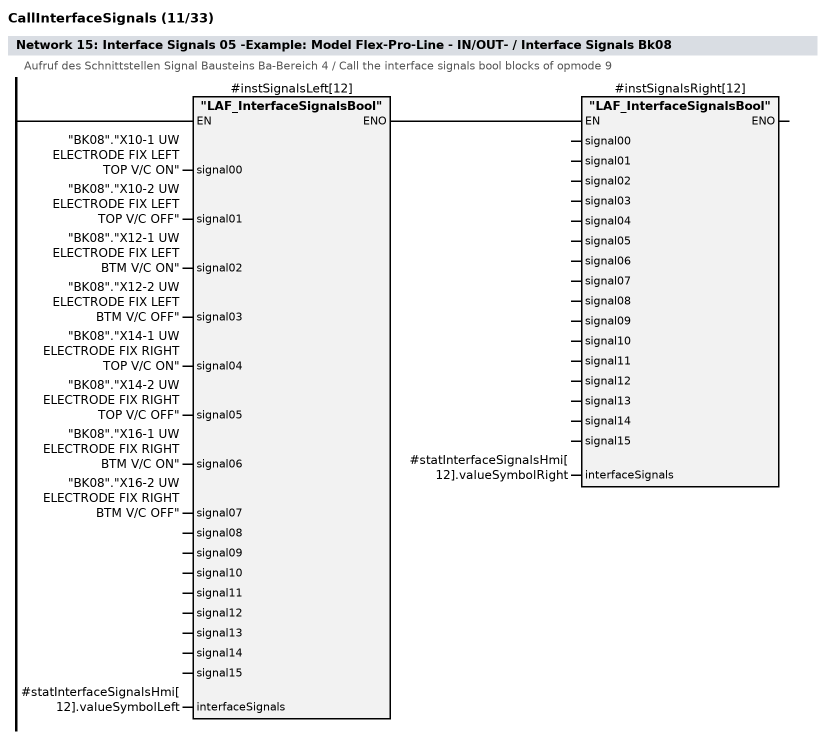
   RUNG wire#powerrail
      #instSignalsLeft[12](signal00 := "BK08"."X10-1 UW ELECTRODE FIX LEFT TOP V/C ON", signal01 := "BK08"."X10-2 UW ELECTRODE FIX LEFT TOP V/C OFF", signal02 := "BK08"."X12-1 UW ELECTRODE FIX LEFT BTM V/C ON", signal03 := "BK08"."X12-2 UW ELECTRODE FIX LEFT BTM V/C OFF", signal04 := "BK08"."X14-1 UW ELECTRODE FIX RIGHT TOP V/C ON", signal05 := "BK08"."X14-2 UW ELECTRODE FIX RIGHT TOP V/C OFF", signal06 := "BK08"."X16-1 UW ELECTRODE FIX RIGHT BTM V/C ON", signal07 := "BK08"."X16-2 UW ELECTRODE FIX RIGHT BTM V/C OFF", signal08 :=, signal09 :=, signal10 :=, signal11 :=, signal12 :=, signal13 :=, signal14 :=, signal15 :=, interfaceSignals := #statInterfaceSignalsHmi[12].valueSymbolLeft)
      #instSignalsRight[12](signal00 :=, signal01 :=, signal02 :=, signal03 :=, signal04 :=, signal05 :=, signal06 :=, signal07 :=, signal08 :=, signal09 :=, signal10 :=, signal11 :=, signal12 :=, signal13 :=, signal14 :=, signal15 :=, interfaceSignals := #statInterfaceSignalsHmi[12].valueSymbolRight)
   END_RUNG
   // the same network as SCL:
   #instSignalsLeft[12](signal00 := "BK08"."X10-1 UW ELECTRODE FIX LEFT TOP V/C ON",   // "LAF_InterfaceSignalsBool"
                        signal01 := "BK08"."X10-2 UW ELECTRODE FIX LEFT TOP V/C OFF",
                        signal02 := "BK08"."X12-1 UW ELECTRODE FIX LEFT BTM V/C ON",
                        signal03 := "BK08"."X12-2 UW ELECTRODE FIX LEFT BTM V/C OFF",
                        signal04 := "BK08"."X14-1 UW ELECTRODE FIX RIGHT TOP V/C ON",
                        signal05 := "BK08"."X14-2 UW ELECTRODE FIX RIGHT TOP V/C OFF",
                        signal06 := "BK08"."X16-1 UW ELECTRODE FIX RIGHT BTM V/C ON",
                        signal07 := "BK08"."X16-2 UW ELECTRODE FIX RIGHT BTM V/C OFF",
                        interfaceSignals := #statInterfaceSignalsHmi[12].valueSymbolLeft,
                        ENO => #_w1);
   IF #_w1 THEN
       #instSignalsRight[12](interfaceSignals := #statInterfaceSignalsHmi[12].valueSymbolRight);   // "LAF_InterfaceSignalsBool"
   END_IF;
END_REGION

REGION Network 16: Interface Signals 06 / Interface Signals Bk09
   // Aufruf des Schnittstellen Signal Bausteins / Call the interface signals bool blocks
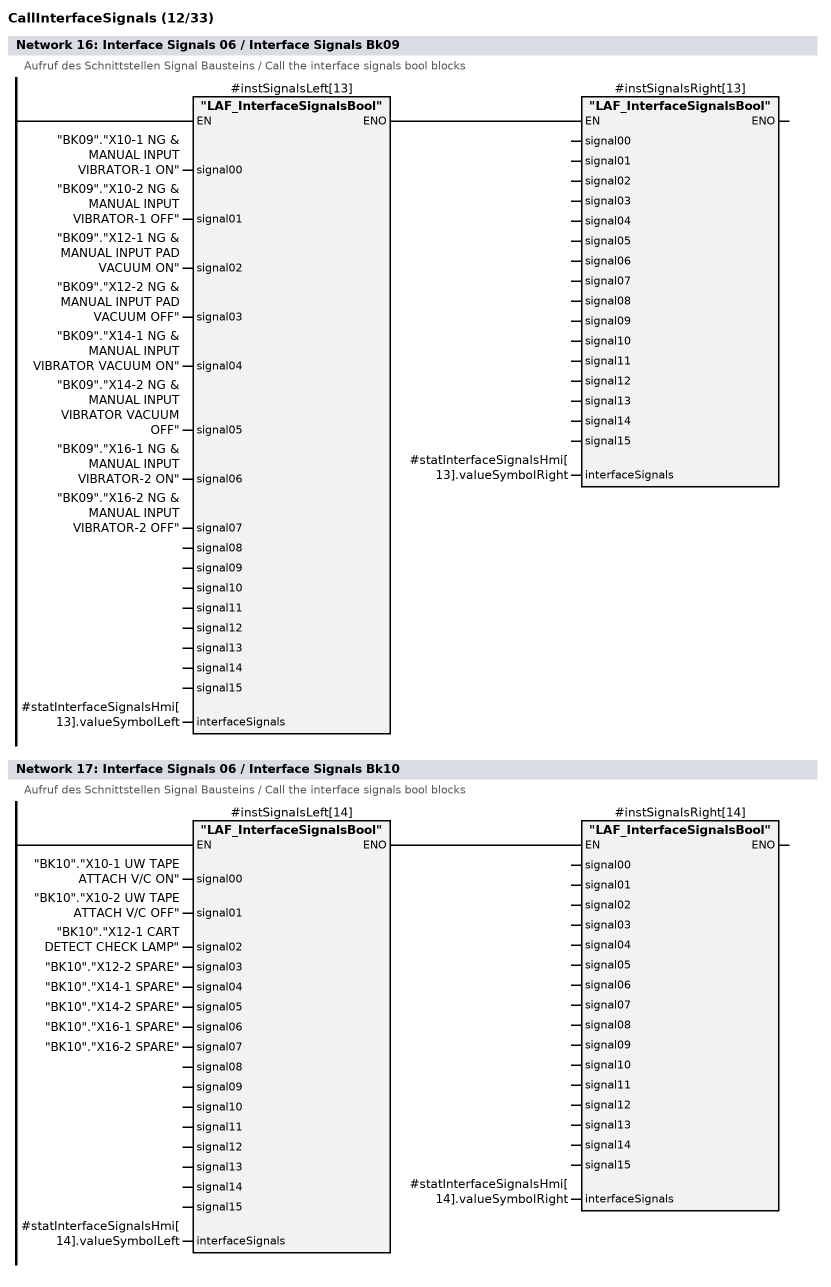
   RUNG wire#powerrail
      #instSignalsLeft[13](signal00 := "BK09"."X10-1 NG & MANUAL INPUT VIBRATOR-1 ON", signal01 := "BK09"."X10-2 NG & MANUAL INPUT VIBRATOR-1 OFF", signal02 := "BK09"."X12-1 NG & MANUAL INPUT PAD VACUUM ON", signal03 := "BK09"."X12-2 NG & MANUAL INPUT PAD VACUUM OFF", signal04 := "BK09"."X14-1 NG & MANUAL INPUT VIBRATOR VACUUM ON", signal05 := "BK09"."X14-2 NG & MANUAL INPUT VIBRATOR VACUUM OFF", signal06 := "BK09"."X16-1 NG & MANUAL INPUT VIBRATOR-2 ON", signal07 := "BK09"."X16-2 NG & MANUAL INPUT VIBRATOR-2 OFF", signal08 :=, signal09 :=, signal10 :=, signal11 :=, signal12 :=, signal13 :=, signal14 :=, signal15 :=, interfaceSignals := #statInterfaceSignalsHmi[13].valueSymbolLeft)
      #instSignalsRight[13](signal00 :=, signal01 :=, signal02 :=, signal03 :=, signal04 :=, signal05 :=, signal06 :=, signal07 :=, signal08 :=, signal09 :=, signal10 :=, signal11 :=, signal12 :=, signal13 :=, signal14 :=, signal15 :=, interfaceSignals := #statInterfaceSignalsHmi[13].valueSymbolRight)
   END_RUNG
   // the same network as SCL:
   #instSignalsLeft[13](signal00 := "BK09"."X10-1 NG & MANUAL INPUT VIBRATOR-1 ON",   // "LAF_InterfaceSignalsBool"
                        signal01 := "BK09"."X10-2 NG & MANUAL INPUT VIBRATOR-1 OFF",
                        signal02 := "BK09"."X12-1 NG & MANUAL INPUT PAD VACUUM ON",
                        signal03 := "BK09"."X12-2 NG & MANUAL INPUT PAD VACUUM OFF",
                        signal04 := "BK09"."X14-1 NG & MANUAL INPUT VIBRATOR VACUUM ON",
                        signal05 := "BK09"."X14-2 NG & MANUAL INPUT VIBRATOR VACUUM OFF",
                        signal06 := "BK09"."X16-1 NG & MANUAL INPUT VIBRATOR-2 ON",
                        signal07 := "BK09"."X16-2 NG & MANUAL INPUT VIBRATOR-2 OFF",
                        interfaceSignals := #statInterfaceSignalsHmi[13].valueSymbolLeft,
                        ENO => #_w1);
   IF #_w1 THEN
       #instSignalsRight[13](interfaceSignals := #statInterfaceSignalsHmi[13].valueSymbolRight);   // "LAF_InterfaceSignalsBool"
   END_IF;
END_REGION

REGION Network 17: Interface Signals 06 / Interface Signals Bk10
   // Aufruf des Schnittstellen Signal Bausteins / Call the interface signals bool blocks
   RUNG wire#powerrail
      #instSignalsLeft[14](signal00 := "BK10"."X10-1 UW TAPE ATTACH V/C ON", signal01 := "BK10"."X10-2 UW TAPE ATTACH V/C OFF", signal02 := "BK10"."X12-1 CART DETECT CHECK LAMP", signal03 := "BK10"."X12-2 SPARE", signal04 := "BK10"."X14-1 SPARE", signal05 := "BK10"."X14-2 SPARE", signal06 := "BK10"."X16-1 SPARE", signal07 := "BK10"."X16-2 SPARE", signal08 :=, signal09 :=, signal10 :=, signal11 :=, signal12 :=, signal13 :=, signal14 :=, signal15 :=, interfaceSignals := #statInterfaceSignalsHmi[14].valueSymbolLeft)
      #instSignalsRight[14](signal00 :=, signal01 :=, signal02 :=, signal03 :=, signal04 :=, signal05 :=, signal06 :=, signal07 :=, signal08 :=, signal09 :=, signal10 :=, signal11 :=, signal12 :=, signal13 :=, signal14 :=, signal15 :=, interfaceSignals := #statInterfaceSignalsHmi[14].valueSymbolRight)
   END_RUNG
   // the same network as SCL:
   #instSignalsLeft[14](signal00 := "BK10"."X10-1 UW TAPE ATTACH V/C ON",   // "LAF_InterfaceSignalsBool"
                        signal01 := "BK10"."X10-2 UW TAPE ATTACH V/C OFF",
                        signal02 := "BK10"."X12-1 CART DETECT CHECK LAMP",
                        signal03 := "BK10"."X12-2 SPARE",
                        signal04 := "BK10"."X14-1 SPARE",
                        signal05 := "BK10"."X14-2 SPARE",
                        signal06 := "BK10"."X16-1 SPARE",
                        signal07 := "BK10"."X16-2 SPARE",
                        interfaceSignals := #statInterfaceSignalsHmi[14].valueSymbolLeft,
                        ENO => #_w1);
   IF #_w1 THEN
       #instSignalsRight[14](interfaceSignals := #statInterfaceSignalsHmi[14].valueSymbolRight);   // "LAF_InterfaceSignalsBool"
   END_IF;
END_REGION

REGION Network 18: Interface Signals 06 / Interface Signals SBK01
   // Aufruf des Schnittstellen Signal Bausteins / Call the interface signals bool blocks
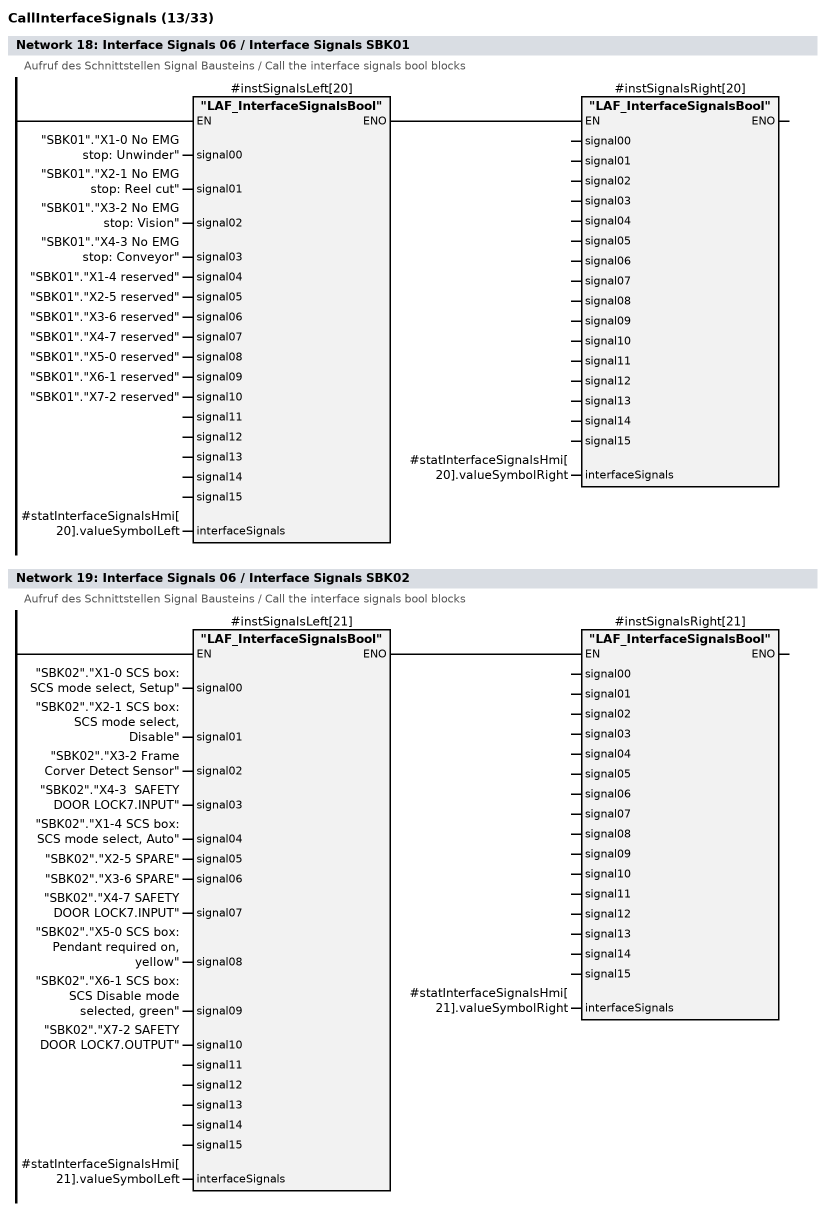
   RUNG wire#powerrail
      #instSignalsLeft[20](signal00 := "SBK01"."X1-0 No EMG stop: Unwinder", signal01 := "SBK01"."X2-1 No EMG stop: Reel cut", signal02 := "SBK01"."X3-2 No EMG stop: Vision", signal03 := "SBK01"."X4-3 No EMG stop: Conveyor", signal04 := "SBK01"."X1-4 reserved", signal05 := "SBK01"."X2-5 reserved", signal06 := "SBK01"."X3-6 reserved", signal07 := "SBK01"."X4-7 reserved", signal08 := "SBK01"."X5-0 reserved", signal09 := "SBK01"."X6-1 reserved", signal10 := "SBK01"."X7-2 reserved", signal11 :=, signal12 :=, signal13 :=, signal14 :=, signal15 :=, interfaceSignals := #statInterfaceSignalsHmi[20].valueSymbolLeft)
      #instSignalsRight[20](signal00 :=, signal01 :=, signal02 :=, signal03 :=, signal04 :=, signal05 :=, signal06 :=, signal07 :=, signal08 :=, signal09 :=, signal10 :=, signal11 :=, signal12 :=, signal13 :=, signal14 :=, signal15 :=, interfaceSignals := #statInterfaceSignalsHmi[20].valueSymbolRight)
   END_RUNG
   // the same network as SCL:
   #instSignalsLeft[20](signal00 := "SBK01"."X1-0 No EMG stop: Unwinder",   // "LAF_InterfaceSignalsBool"
                        signal01 := "SBK01"."X2-1 No EMG stop: Reel cut",
                        signal02 := "SBK01"."X3-2 No EMG stop: Vision",
                        signal03 := "SBK01"."X4-3 No EMG stop: Conveyor",
                        signal04 := "SBK01"."X1-4 reserved",
                        signal05 := "SBK01"."X2-5 reserved",
                        signal06 := "SBK01"."X3-6 reserved",
                        signal07 := "SBK01"."X4-7 reserved",
                        signal08 := "SBK01"."X5-0 reserved",
                        signal09 := "SBK01"."X6-1 reserved",
                        signal10 := "SBK01"."X7-2 reserved",
                        interfaceSignals := #statInterfaceSignalsHmi[20].valueSymbolLeft,
                        ENO => #_w1);
   IF #_w1 THEN
       #instSignalsRight[20](interfaceSignals := #statInterfaceSignalsHmi[20].valueSymbolRight);   // "LAF_InterfaceSignalsBool"
   END_IF;
END_REGION

REGION Network 19: Interface Signals 06 / Interface Signals SBK02
   // Aufruf des Schnittstellen Signal Bausteins / Call the interface signals bool blocks
   RUNG wire#powerrail
      #instSignalsLeft[21](signal00 := "SBK02"."X1-0 SCS box: SCS mode select, Setup", signal01 := "SBK02"."X2-1 SCS box: SCS mode select, Disable", signal02 := "SBK02"."X3-2 Frame Corver Detect Sensor", signal03 := "SBK02"."X4-3  SAFETY DOOR LOCK7.INPUT", signal04 := "SBK02"."X1-4 SCS box: SCS mode select, Auto", signal05 := "SBK02"."X2-5 SPARE", signal06 := "SBK02"."X3-6 SPARE", signal07 := "SBK02"."X4-7 SAFETY DOOR LOCK7.INPUT", signal08 := "SBK02"."X5-0 SCS box: Pendant required on, yellow", signal09 := "SBK02"."X6-1 SCS box: SCS Disable mode selected, green", signal10 := "SBK02"."X7-2 SAFETY DOOR LOCK7.OUTPUT", signal11 :=, signal12 :=, signal13 :=, signal14 :=, signal15 :=, interfaceSignals := #statInterfaceSignalsHmi[21].valueSymbolLeft)
      #instSignalsRight[21](signal00 :=, signal01 :=, signal02 :=, signal03 :=, signal04 :=, signal05 :=, signal06 :=, signal07 :=, signal08 :=, signal09 :=, signal10 :=, signal11 :=, signal12 :=, signal13 :=, signal14 :=, signal15 :=, interfaceSignals := #statInterfaceSignalsHmi[21].valueSymbolRight)
   END_RUNG
   // the same network as SCL:
   #instSignalsLeft[21](signal00 := "SBK02"."X1-0 SCS box: SCS mode select, Setup",   // "LAF_InterfaceSignalsBool"
                        signal01 := "SBK02"."X2-1 SCS box: SCS mode select, Disable",
                        signal02 := "SBK02"."X3-2 Frame Corver Detect Sensor",
                        signal03 := "SBK02"."X4-3  SAFETY DOOR LOCK7.INPUT",
                        signal04 := "SBK02"."X1-4 SCS box: SCS mode select, Auto",
                        signal05 := "SBK02"."X2-5 SPARE",
                        signal06 := "SBK02"."X3-6 SPARE",
                        signal07 := "SBK02"."X4-7 SAFETY DOOR LOCK7.INPUT",
                        signal08 := "SBK02"."X5-0 SCS box: Pendant required on, yellow",
                        signal09 := "SBK02"."X6-1 SCS box: SCS Disable mode selected, green",
                        signal10 := "SBK02"."X7-2 SAFETY DOOR LOCK7.OUTPUT",
                        interfaceSignals := #statInterfaceSignalsHmi[21].valueSymbolLeft,
                        ENO => #_w1);
   IF #_w1 THEN
       #instSignalsRight[21](interfaceSignals := #statInterfaceSignalsHmi[21].valueSymbolRight);   // "LAF_InterfaceSignalsBool"
   END_IF;
END_REGION

REGION Network 20: Interface Signals 06 / Interface Signals SBK03
   // Aufruf des Schnittstellen Signal Bausteins / Call the interface signals bool blocks
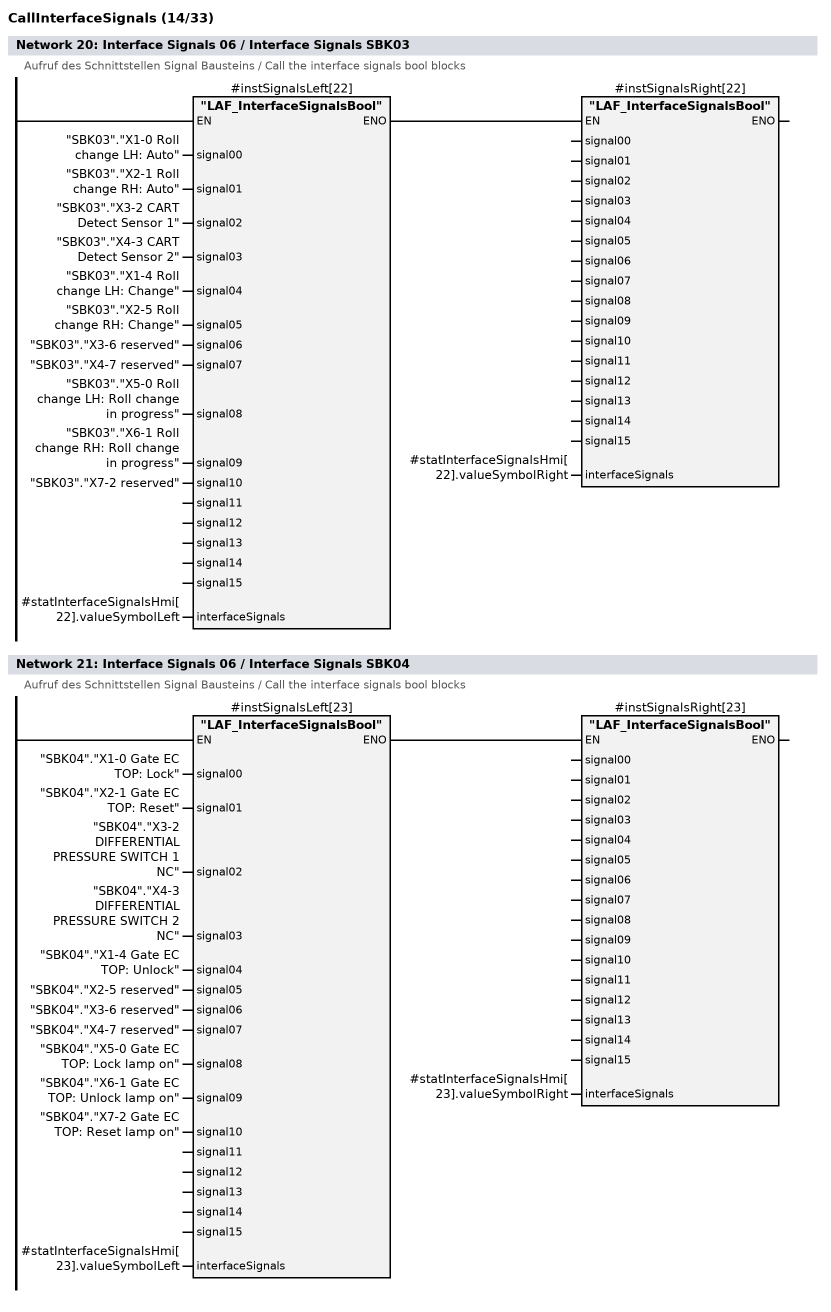
   RUNG wire#powerrail
      #instSignalsLeft[22](signal00 := "SBK03"."X1-0 Roll change LH: Auto", signal01 := "SBK03"."X2-1 Roll change RH: Auto", signal02 := "SBK03"."X3-2 CART Detect Sensor 1", signal03 := "SBK03"."X4-3 CART Detect Sensor 2", signal04 := "SBK03"."X1-4 Roll change LH: Change", signal05 := "SBK03"."X2-5 Roll change RH: Change", signal06 := "SBK03"."X3-6 reserved", signal07 := "SBK03"."X4-7 reserved", signal08 := "SBK03"."X5-0 Roll change LH: Roll change in progress", signal09 := "SBK03"."X6-1 Roll change RH: Roll change in progress", signal10 := "SBK03"."X7-2 reserved", signal11 :=, signal12 :=, signal13 :=, signal14 :=, signal15 :=, interfaceSignals := #statInterfaceSignalsHmi[22].valueSymbolLeft)
      #instSignalsRight[22](signal00 :=, signal01 :=, signal02 :=, signal03 :=, signal04 :=, signal05 :=, signal06 :=, signal07 :=, signal08 :=, signal09 :=, signal10 :=, signal11 :=, signal12 :=, signal13 :=, signal14 :=, signal15 :=, interfaceSignals := #statInterfaceSignalsHmi[22].valueSymbolRight)
   END_RUNG
   // the same network as SCL:
   #instSignalsLeft[22](signal00 := "SBK03"."X1-0 Roll change LH: Auto",   // "LAF_InterfaceSignalsBool"
                        signal01 := "SBK03"."X2-1 Roll change RH: Auto",
                        signal02 := "SBK03"."X3-2 CART Detect Sensor 1",
                        signal03 := "SBK03"."X4-3 CART Detect Sensor 2",
                        signal04 := "SBK03"."X1-4 Roll change LH: Change",
                        signal05 := "SBK03"."X2-5 Roll change RH: Change",
                        signal06 := "SBK03"."X3-6 reserved",
                        signal07 := "SBK03"."X4-7 reserved",
                        signal08 := "SBK03"."X5-0 Roll change LH: Roll change in progress",
                        signal09 := "SBK03"."X6-1 Roll change RH: Roll change in progress",
                        signal10 := "SBK03"."X7-2 reserved",
                        interfaceSignals := #statInterfaceSignalsHmi[22].valueSymbolLeft,
                        ENO => #_w1);
   IF #_w1 THEN
       #instSignalsRight[22](interfaceSignals := #statInterfaceSignalsHmi[22].valueSymbolRight);   // "LAF_InterfaceSignalsBool"
   END_IF;
END_REGION

REGION Network 21: Interface Signals 06 / Interface Signals SBK04
   // Aufruf des Schnittstellen Signal Bausteins / Call the interface signals bool blocks
   RUNG wire#powerrail
      #instSignalsLeft[23](signal00 := "SBK04"."X1-0 Gate EC TOP: Lock", signal01 := "SBK04"."X2-1 Gate EC TOP: Reset", signal02 := "SBK04"."X3-2 DIFFERENTIAL PRESSURE SWITCH 1 NC", signal03 := "SBK04"."X4-3 DIFFERENTIAL PRESSURE SWITCH 2 NC", signal04 := "SBK04"."X1-4 Gate EC TOP: Unlock", signal05 := "SBK04"."X2-5 reserved", signal06 := "SBK04"."X3-6 reserved", signal07 := "SBK04"."X4-7 reserved", signal08 := "SBK04"."X5-0 Gate EC TOP: Lock lamp on", signal09 := "SBK04"."X6-1 Gate EC TOP: Unlock lamp on", signal10 := "SBK04"."X7-2 Gate EC TOP: Reset lamp on", signal11 :=, signal12 :=, signal13 :=, signal14 :=, signal15 :=, interfaceSignals := #statInterfaceSignalsHmi[23].valueSymbolLeft)
      #instSignalsRight[23](signal00 :=, signal01 :=, signal02 :=, signal03 :=, signal04 :=, signal05 :=, signal06 :=, signal07 :=, signal08 :=, signal09 :=, signal10 :=, signal11 :=, signal12 :=, signal13 :=, signal14 :=, signal15 :=, interfaceSignals := #statInterfaceSignalsHmi[23].valueSymbolRight)
   END_RUNG
   // the same network as SCL:
   #instSignalsLeft[23](signal00 := "SBK04"."X1-0 Gate EC TOP: Lock",   // "LAF_InterfaceSignalsBool"
                        signal01 := "SBK04"."X2-1 Gate EC TOP: Reset",
                        signal02 := "SBK04"."X3-2 DIFFERENTIAL PRESSURE SWITCH 1 NC",
                        signal03 := "SBK04"."X4-3 DIFFERENTIAL PRESSURE SWITCH 2 NC",
                        signal04 := "SBK04"."X1-4 Gate EC TOP: Unlock",
                        signal05 := "SBK04"."X2-5 reserved",
                        signal06 := "SBK04"."X3-6 reserved",
                        signal07 := "SBK04"."X4-7 reserved",
                        signal08 := "SBK04"."X5-0 Gate EC TOP: Lock lamp on",
                        signal09 := "SBK04"."X6-1 Gate EC TOP: Unlock lamp on",
                        signal10 := "SBK04"."X7-2 Gate EC TOP: Reset lamp on",
                        interfaceSignals := #statInterfaceSignalsHmi[23].valueSymbolLeft,
                        ENO => #_w1);
   IF #_w1 THEN
       #instSignalsRight[23](interfaceSignals := #statInterfaceSignalsHmi[23].valueSymbolRight);   // "LAF_InterfaceSignalsBool"
   END_IF;
END_REGION

REGION Network 22: Interface Signals 06 / Interface Signals SBK05
   // Aufruf des Schnittstellen Signal Bausteins / Call the interface signals bool blocks
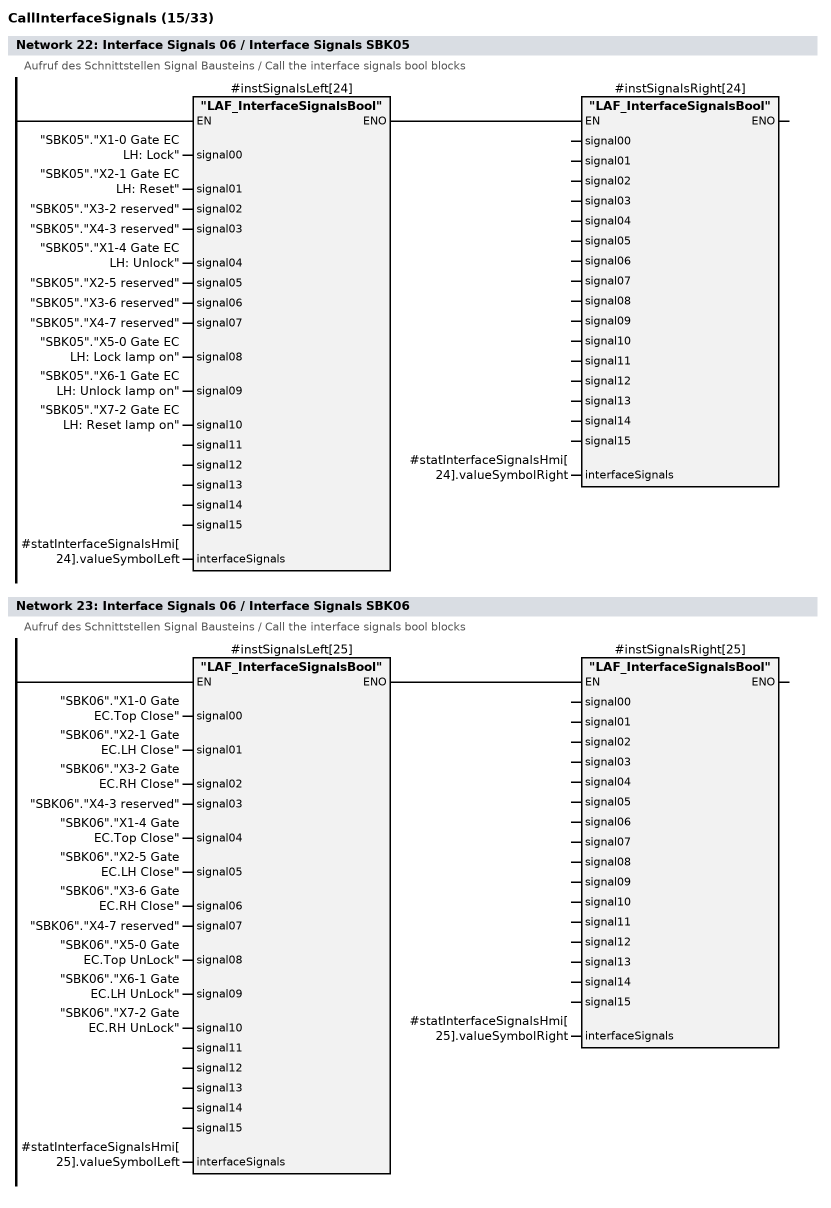
   RUNG wire#powerrail
      #instSignalsLeft[24](signal00 := "SBK05"."X1-0 Gate EC LH: Lock", signal01 := "SBK05"."X2-1 Gate EC LH: Reset", signal02 := "SBK05"."X3-2 reserved", signal03 := "SBK05"."X4-3 reserved", signal04 := "SBK05"."X1-4 Gate EC LH: Unlock", signal05 := "SBK05"."X2-5 reserved", signal06 := "SBK05"."X3-6 reserved", signal07 := "SBK05"."X4-7 reserved", signal08 := "SBK05"."X5-0 Gate EC LH: Lock lamp on", signal09 := "SBK05"."X6-1 Gate EC LH: Unlock lamp on", signal10 := "SBK05"."X7-2 Gate EC LH: Reset lamp on", signal11 :=, signal12 :=, signal13 :=, signal14 :=, signal15 :=, interfaceSignals := #statInterfaceSignalsHmi[24].valueSymbolLeft)
      #instSignalsRight[24](signal00 :=, signal01 :=, signal02 :=, signal03 :=, signal04 :=, signal05 :=, signal06 :=, signal07 :=, signal08 :=, signal09 :=, signal10 :=, signal11 :=, signal12 :=, signal13 :=, signal14 :=, signal15 :=, interfaceSignals := #statInterfaceSignalsHmi[24].valueSymbolRight)
   END_RUNG
   // the same network as SCL:
   #instSignalsLeft[24](signal00 := "SBK05"."X1-0 Gate EC LH: Lock",   // "LAF_InterfaceSignalsBool"
                        signal01 := "SBK05"."X2-1 Gate EC LH: Reset",
                        signal02 := "SBK05"."X3-2 reserved",
                        signal03 := "SBK05"."X4-3 reserved",
                        signal04 := "SBK05"."X1-4 Gate EC LH: Unlock",
                        signal05 := "SBK05"."X2-5 reserved",
                        signal06 := "SBK05"."X3-6 reserved",
                        signal07 := "SBK05"."X4-7 reserved",
                        signal08 := "SBK05"."X5-0 Gate EC LH: Lock lamp on",
                        signal09 := "SBK05"."X6-1 Gate EC LH: Unlock lamp on",
                        signal10 := "SBK05"."X7-2 Gate EC LH: Reset lamp on",
                        interfaceSignals := #statInterfaceSignalsHmi[24].valueSymbolLeft,
                        ENO => #_w1);
   IF #_w1 THEN
       #instSignalsRight[24](interfaceSignals := #statInterfaceSignalsHmi[24].valueSymbolRight);   // "LAF_InterfaceSignalsBool"
   END_IF;
END_REGION

REGION Network 23: Interface Signals 06 / Interface Signals SBK06
   // Aufruf des Schnittstellen Signal Bausteins / Call the interface signals bool blocks
   RUNG wire#powerrail
      #instSignalsLeft[25](signal00 := "SBK06"."X1-0 Gate EC.Top Close", signal01 := "SBK06"."X2-1 Gate EC.LH Close", signal02 := "SBK06"."X3-2 Gate EC.RH Close", signal03 := "SBK06"."X4-3 reserved", signal04 := "SBK06"."X1-4 Gate EC.Top Close", signal05 := "SBK06"."X2-5 Gate EC.LH Close", signal06 := "SBK06"."X3-6 Gate EC.RH Close", signal07 := "SBK06"."X4-7 reserved", signal08 := "SBK06"."X5-0 Gate EC.Top UnLock", signal09 := "SBK06"."X6-1 Gate EC.LH UnLock", signal10 := "SBK06"."X7-2 Gate EC.RH UnLock", signal11 :=, signal12 :=, signal13 :=, signal14 :=, signal15 :=, interfaceSignals := #statInterfaceSignalsHmi[25].valueSymbolLeft)
      #instSignalsRight[25](signal00 :=, signal01 :=, signal02 :=, signal03 :=, signal04 :=, signal05 :=, signal06 :=, signal07 :=, signal08 :=, signal09 :=, signal10 :=, signal11 :=, signal12 :=, signal13 :=, signal14 :=, signal15 :=, interfaceSignals := #statInterfaceSignalsHmi[25].valueSymbolRight)
   END_RUNG
   // the same network as SCL:
   #instSignalsLeft[25](signal00 := "SBK06"."X1-0 Gate EC.Top Close",   // "LAF_InterfaceSignalsBool"
                        signal01 := "SBK06"."X2-1 Gate EC.LH Close",
                        signal02 := "SBK06"."X3-2 Gate EC.RH Close",
                        signal03 := "SBK06"."X4-3 reserved",
                        signal04 := "SBK06"."X1-4 Gate EC.Top Close",
                        signal05 := "SBK06"."X2-5 Gate EC.LH Close",
                        signal06 := "SBK06"."X3-6 Gate EC.RH Close",
                        signal07 := "SBK06"."X4-7 reserved",
                        signal08 := "SBK06"."X5-0 Gate EC.Top UnLock",
                        signal09 := "SBK06"."X6-1 Gate EC.LH UnLock",
                        signal10 := "SBK06"."X7-2 Gate EC.RH UnLock",
                        interfaceSignals := #statInterfaceSignalsHmi[25].valueSymbolLeft,
                        ENO => #_w1);
   IF #_w1 THEN
       #instSignalsRight[25](interfaceSignals := #statInterfaceSignalsHmi[25].valueSymbolRight);   // "LAF_InterfaceSignalsBool"
   END_IF;
END_REGION

REGION Network 24: Interface Signals 06 / Interface Signals SBK07
   // Aufruf des Schnittstellen Signal Bausteins / Call the interface signals bool blocks
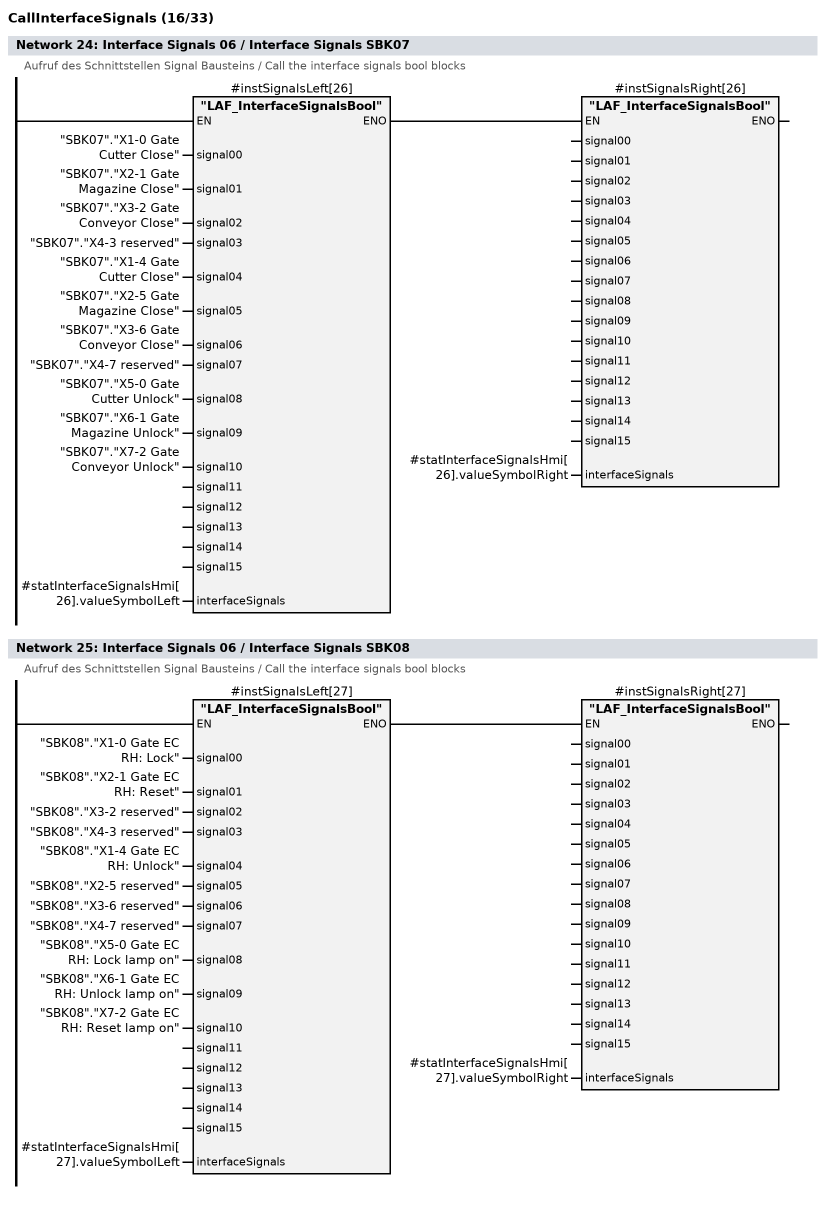
   RUNG wire#powerrail
      #instSignalsLeft[26](signal00 := "SBK07"."X1-0 Gate Cutter Close", signal01 := "SBK07"."X2-1 Gate Magazine Close", signal02 := "SBK07"."X3-2 Gate Conveyor Close", signal03 := "SBK07"."X4-3 reserved", signal04 := "SBK07"."X1-4 Gate Cutter Close", signal05 := "SBK07"."X2-5 Gate Magazine Close", signal06 := "SBK07"."X3-6 Gate Conveyor Close", signal07 := "SBK07"."X4-7 reserved", signal08 := "SBK07"."X5-0 Gate Cutter Unlock", signal09 := "SBK07"."X6-1 Gate Magazine Unlock", signal10 := "SBK07"."X7-2 Gate Conveyor Unlock", signal11 :=, signal12 :=, signal13 :=, signal14 :=, signal15 :=, interfaceSignals := #statInterfaceSignalsHmi[26].valueSymbolLeft)
      #instSignalsRight[26](signal00 :=, signal01 :=, signal02 :=, signal03 :=, signal04 :=, signal05 :=, signal06 :=, signal07 :=, signal08 :=, signal09 :=, signal10 :=, signal11 :=, signal12 :=, signal13 :=, signal14 :=, signal15 :=, interfaceSignals := #statInterfaceSignalsHmi[26].valueSymbolRight)
   END_RUNG
   // the same network as SCL:
   #instSignalsLeft[26](signal00 := "SBK07"."X1-0 Gate Cutter Close",   // "LAF_InterfaceSignalsBool"
                        signal01 := "SBK07"."X2-1 Gate Magazine Close",
                        signal02 := "SBK07"."X3-2 Gate Conveyor Close",
                        signal03 := "SBK07"."X4-3 reserved",
                        signal04 := "SBK07"."X1-4 Gate Cutter Close",
                        signal05 := "SBK07"."X2-5 Gate Magazine Close",
                        signal06 := "SBK07"."X3-6 Gate Conveyor Close",
                        signal07 := "SBK07"."X4-7 reserved",
                        signal08 := "SBK07"."X5-0 Gate Cutter Unlock",
                        signal09 := "SBK07"."X6-1 Gate Magazine Unlock",
                        signal10 := "SBK07"."X7-2 Gate Conveyor Unlock",
                        interfaceSignals := #statInterfaceSignalsHmi[26].valueSymbolLeft,
                        ENO => #_w1);
   IF #_w1 THEN
       #instSignalsRight[26](interfaceSignals := #statInterfaceSignalsHmi[26].valueSymbolRight);   // "LAF_InterfaceSignalsBool"
   END_IF;
END_REGION

REGION Network 25: Interface Signals 06 / Interface Signals SBK08
   // Aufruf des Schnittstellen Signal Bausteins / Call the interface signals bool blocks
   RUNG wire#powerrail
      #instSignalsLeft[27](signal00 := "SBK08"."X1-0 Gate EC RH: Lock", signal01 := "SBK08"."X2-1 Gate EC RH: Reset", signal02 := "SBK08"."X3-2 reserved", signal03 := "SBK08"."X4-3 reserved", signal04 := "SBK08"."X1-4 Gate EC RH: Unlock", signal05 := "SBK08"."X2-5 reserved", signal06 := "SBK08"."X3-6 reserved", signal07 := "SBK08"."X4-7 reserved", signal08 := "SBK08"."X5-0 Gate EC RH: Lock lamp on", signal09 := "SBK08"."X6-1 Gate EC RH: Unlock lamp on", signal10 := "SBK08"."X7-2 Gate EC RH: Reset lamp on", signal11 :=, signal12 :=, signal13 :=, signal14 :=, signal15 :=, interfaceSignals := #statInterfaceSignalsHmi[27].valueSymbolLeft)
      #instSignalsRight[27](signal00 :=, signal01 :=, signal02 :=, signal03 :=, signal04 :=, signal05 :=, signal06 :=, signal07 :=, signal08 :=, signal09 :=, signal10 :=, signal11 :=, signal12 :=, signal13 :=, signal14 :=, signal15 :=, interfaceSignals := #statInterfaceSignalsHmi[27].valueSymbolRight)
   END_RUNG
   // the same network as SCL:
   #instSignalsLeft[27](signal00 := "SBK08"."X1-0 Gate EC RH: Lock",   // "LAF_InterfaceSignalsBool"
                        signal01 := "SBK08"."X2-1 Gate EC RH: Reset",
                        signal02 := "SBK08"."X3-2 reserved",
                        signal03 := "SBK08"."X4-3 reserved",
                        signal04 := "SBK08"."X1-4 Gate EC RH: Unlock",
                        signal05 := "SBK08"."X2-5 reserved",
                        signal06 := "SBK08"."X3-6 reserved",
                        signal07 := "SBK08"."X4-7 reserved",
                        signal08 := "SBK08"."X5-0 Gate EC RH: Lock lamp on",
                        signal09 := "SBK08"."X6-1 Gate EC RH: Unlock lamp on",
                        signal10 := "SBK08"."X7-2 Gate EC RH: Reset lamp on",
                        interfaceSignals := #statInterfaceSignalsHmi[27].valueSymbolLeft,
                        ENO => #_w1);
   IF #_w1 THEN
       #instSignalsRight[27](interfaceSignals := #statInterfaceSignalsHmi[27].valueSymbolRight);   // "LAF_InterfaceSignalsBool"
   END_IF;
END_REGION

REGION Network 26: Interface Signals 06 / Interface Signals SBK09
   // Aufruf des Schnittstellen Signal Bausteins / Call the interface signals bool blocks
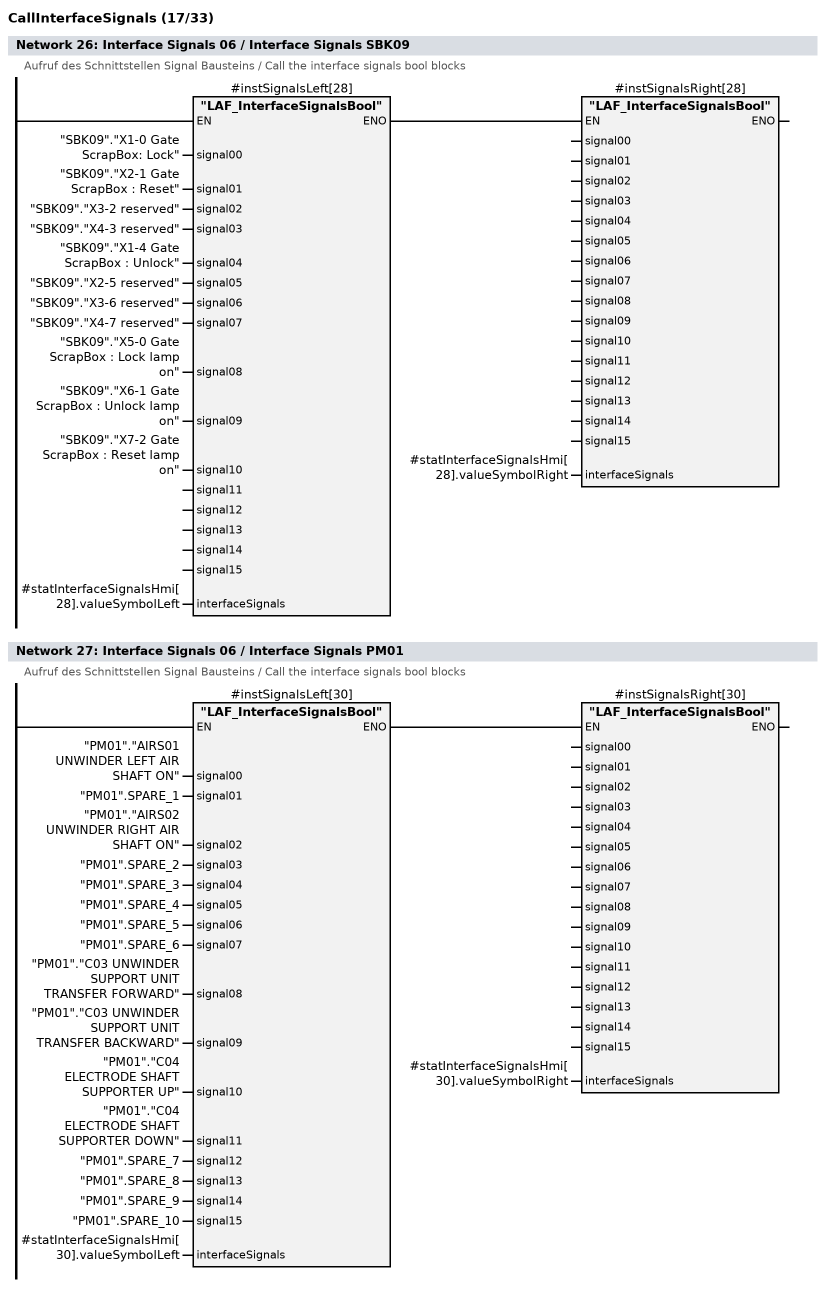
   RUNG wire#powerrail
      #instSignalsLeft[28](signal00 := "SBK09"."X1-0 Gate ScrapBox: Lock", signal01 := "SBK09"."X2-1 Gate ScrapBox : Reset", signal02 := "SBK09"."X3-2 reserved", signal03 := "SBK09"."X4-3 reserved", signal04 := "SBK09"."X1-4 Gate ScrapBox : Unlock", signal05 := "SBK09"."X2-5 reserved", signal06 := "SBK09"."X3-6 reserved", signal07 := "SBK09"."X4-7 reserved", signal08 := "SBK09"."X5-0 Gate ScrapBox : Lock lamp on", signal09 := "SBK09"."X6-1 Gate ScrapBox : Unlock lamp on", signal10 := "SBK09"."X7-2 Gate ScrapBox : Reset lamp on", signal11 :=, signal12 :=, signal13 :=, signal14 :=, signal15 :=, interfaceSignals := #statInterfaceSignalsHmi[28].valueSymbolLeft)
      #instSignalsRight[28](signal00 :=, signal01 :=, signal02 :=, signal03 :=, signal04 :=, signal05 :=, signal06 :=, signal07 :=, signal08 :=, signal09 :=, signal10 :=, signal11 :=, signal12 :=, signal13 :=, signal14 :=, signal15 :=, interfaceSignals := #statInterfaceSignalsHmi[28].valueSymbolRight)
   END_RUNG
   // the same network as SCL:
   #instSignalsLeft[28](signal00 := "SBK09"."X1-0 Gate ScrapBox: Lock",   // "LAF_InterfaceSignalsBool"
                        signal01 := "SBK09"."X2-1 Gate ScrapBox : Reset",
                        signal02 := "SBK09"."X3-2 reserved",
                        signal03 := "SBK09"."X4-3 reserved",
                        signal04 := "SBK09"."X1-4 Gate ScrapBox : Unlock",
                        signal05 := "SBK09"."X2-5 reserved",
                        signal06 := "SBK09"."X3-6 reserved",
                        signal07 := "SBK09"."X4-7 reserved",
                        signal08 := "SBK09"."X5-0 Gate ScrapBox : Lock lamp on",
                        signal09 := "SBK09"."X6-1 Gate ScrapBox : Unlock lamp on",
                        signal10 := "SBK09"."X7-2 Gate ScrapBox : Reset lamp on",
                        interfaceSignals := #statInterfaceSignalsHmi[28].valueSymbolLeft,
                        ENO => #_w1);
   IF #_w1 THEN
       #instSignalsRight[28](interfaceSignals := #statInterfaceSignalsHmi[28].valueSymbolRight);   // "LAF_InterfaceSignalsBool"
   END_IF;
END_REGION

REGION Network 27: Interface Signals 06 / Interface Signals PM01
   // Aufruf des Schnittstellen Signal Bausteins / Call the interface signals bool blocks
   RUNG wire#powerrail
      #instSignalsLeft[30](signal00 := "PM01"."AIRS01 UNWINDER LEFT AIR SHAFT ON", signal01 := "PM01".SPARE_1, signal02 := "PM01"."AIRS02 UNWINDER RIGHT AIR SHAFT ON", signal03 := "PM01".SPARE_2, signal04 := "PM01".SPARE_3, signal05 := "PM01".SPARE_4, signal06 := "PM01".SPARE_5, signal07 := "PM01".SPARE_6, signal08 := "PM01"."C03 UNWINDER SUPPORT UNIT TRANSFER FORWARD", signal09 := "PM01"."C03 UNWINDER SUPPORT UNIT TRANSFER BACKWARD", signal10 := "PM01"."C04 ELECTRODE SHAFT SUPPORTER UP", signal11 := "PM01"."C04 ELECTRODE SHAFT SUPPORTER DOWN", signal12 := "PM01".SPARE_7, signal13 := "PM01".SPARE_8, signal14 := "PM01".SPARE_9, signal15 := "PM01".SPARE_10, interfaceSignals := #statInterfaceSignalsHmi[30].valueSymbolLeft)
      #instSignalsRight[30](signal00 :=, signal01 :=, signal02 :=, signal03 :=, signal04 :=, signal05 :=, signal06 :=, signal07 :=, signal08 :=, signal09 :=, signal10 :=, signal11 :=, signal12 :=, signal13 :=, signal14 :=, signal15 :=, interfaceSignals := #statInterfaceSignalsHmi[30].valueSymbolRight)
   END_RUNG
   // the same network as SCL:
   #instSignalsLeft[30](signal00 := "PM01"."AIRS01 UNWINDER LEFT AIR SHAFT ON",   // "LAF_InterfaceSignalsBool"
                        signal01 := "PM01".SPARE_1,
                        signal02 := "PM01"."AIRS02 UNWINDER RIGHT AIR SHAFT ON",
                        signal03 := "PM01".SPARE_2,
                        signal04 := "PM01".SPARE_3,
                        signal05 := "PM01".SPARE_4,
                        signal06 := "PM01".SPARE_5,
                        signal07 := "PM01".SPARE_6,
                        signal08 := "PM01"."C03 UNWINDER SUPPORT UNIT TRANSFER FORWARD",
                        signal09 := "PM01"."C03 UNWINDER SUPPORT UNIT TRANSFER BACKWARD",
                        signal10 := "PM01"."C04 ELECTRODE SHAFT SUPPORTER UP",
                        signal11 := "PM01"."C04 ELECTRODE SHAFT SUPPORTER DOWN",
                        signal12 := "PM01".SPARE_7,
                        signal13 := "PM01".SPARE_8,
                        signal14 := "PM01".SPARE_9,
                        signal15 := "PM01".SPARE_10,
                        interfaceSignals := #statInterfaceSignalsHmi[30].valueSymbolLeft,
                        ENO => #_w1);
   IF #_w1 THEN
       #instSignalsRight[30](interfaceSignals := #statInterfaceSignalsHmi[30].valueSymbolRight);   // "LAF_InterfaceSignalsBool"
   END_IF;
END_REGION

REGION Network 28: Interface Signals 06 / Interface Signals PM02
   // Aufruf des Schnittstellen Signal Bausteins / Call the interface signals bool blocks
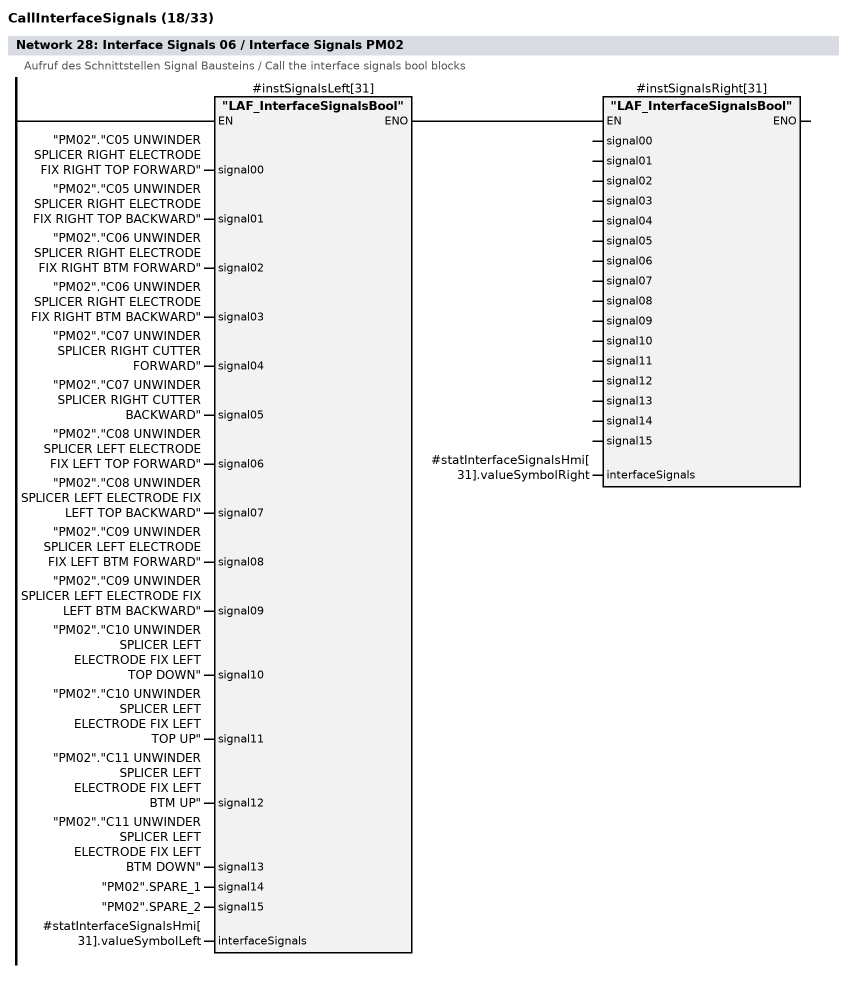
   RUNG wire#powerrail
      #instSignalsLeft[31](signal00 := "PM02"."C05 UNWINDER SPLICER RIGHT ELECTRODE FIX RIGHT TOP FORWARD", signal01 := "PM02"."C05 UNWINDER SPLICER RIGHT ELECTRODE FIX RIGHT TOP BACKWARD", signal02 := "PM02"."C06 UNWINDER SPLICER RIGHT ELECTRODE FIX RIGHT BTM FORWARD", signal03 := "PM02"."C06 UNWINDER SPLICER RIGHT ELECTRODE FIX RIGHT BTM BACKWARD", signal04 := "PM02"."C07 UNWINDER SPLICER RIGHT CUTTER FORWARD", signal05 := "PM02"."C07 UNWINDER SPLICER RIGHT CUTTER BACKWARD", signal06 := "PM02"."C08 UNWINDER SPLICER LEFT ELECTRODE FIX LEFT TOP FORWARD", signal07 := "PM02"."C08 UNWINDER SPLICER LEFT ELECTRODE FIX LEFT TOP BACKWARD", signal08 := "PM02"."C09 UNWINDER SPLICER LEFT ELECTRODE FIX LEFT BTM FORWARD", signal09 := "PM02"."C09 UNWINDER SPLICER LEFT ELECTRODE FIX LEFT BTM BACKWARD", signal10 := "PM02"."C10 UNWINDER SPLICER LEFT ELECTRODE FIX LEFT TOP DOWN", signal11 := "PM02"."C10 UNWINDER SPLICER LEFT ELECTRODE FIX LEFT TOP UP", signal12 := "PM02"."C11 UNWINDER SPLICER LEFT ELECTRODE FIX LEFT BTM UP", signal13 := "PM02"."C11 UNWINDER SPLICER LEFT ELECTRODE FIX LEFT BTM DOWN", signal14 := "PM02".SPARE_1, signal15 := "PM02".SPARE_2, interfaceSignals := #statInterfaceSignalsHmi[31].valueSymbolLeft)
      #instSignalsRight[31](signal00 :=, signal01 :=, signal02 :=, signal03 :=, signal04 :=, signal05 :=, signal06 :=, signal07 :=, signal08 :=, signal09 :=, signal10 :=, signal11 :=, signal12 :=, signal13 :=, signal14 :=, signal15 :=, interfaceSignals := #statInterfaceSignalsHmi[31].valueSymbolRight)
   END_RUNG
   // the same network as SCL:
   #instSignalsLeft[31](signal00 := "PM02"."C05 UNWINDER SPLICER RIGHT ELECTRODE FIX RIGHT TOP FORWARD",   // "LAF_InterfaceSignalsBool"
                        signal01 := "PM02"."C05 UNWINDER SPLICER RIGHT ELECTRODE FIX RIGHT TOP BACKWARD",
                        signal02 := "PM02"."C06 UNWINDER SPLICER RIGHT ELECTRODE FIX RIGHT BTM FORWARD",
                        signal03 := "PM02"."C06 UNWINDER SPLICER RIGHT ELECTRODE FIX RIGHT BTM BACKWARD",
                        signal04 := "PM02"."C07 UNWINDER SPLICER RIGHT CUTTER FORWARD",
                        signal05 := "PM02"."C07 UNWINDER SPLICER RIGHT CUTTER BACKWARD",
                        signal06 := "PM02"."C08 UNWINDER SPLICER LEFT ELECTRODE FIX LEFT TOP FORWARD",
                        signal07 := "PM02"."C08 UNWINDER SPLICER LEFT ELECTRODE FIX LEFT TOP BACKWARD",
                        signal08 := "PM02"."C09 UNWINDER SPLICER LEFT ELECTRODE FIX LEFT BTM FORWARD",
                        signal09 := "PM02"."C09 UNWINDER SPLICER LEFT ELECTRODE FIX LEFT BTM BACKWARD",
                        signal10 := "PM02"."C10 UNWINDER SPLICER LEFT ELECTRODE FIX LEFT TOP DOWN",
                        signal11 := "PM02"."C10 UNWINDER SPLICER LEFT ELECTRODE FIX LEFT TOP UP",
                        signal12 := "PM02"."C11 UNWINDER SPLICER LEFT ELECTRODE FIX LEFT BTM UP",
                        signal13 := "PM02"."C11 UNWINDER SPLICER LEFT ELECTRODE FIX LEFT BTM DOWN",
                        signal14 := "PM02".SPARE_1,
                        signal15 := "PM02".SPARE_2,
                        interfaceSignals := #statInterfaceSignalsHmi[31].valueSymbolLeft,
                        ENO => #_w1);
   IF #_w1 THEN
       #instSignalsRight[31](interfaceSignals := #statInterfaceSignalsHmi[31].valueSymbolRight);   // "LAF_InterfaceSignalsBool"
   END_IF;
END_REGION

REGION Network 29: Interface Signals 06 / Interface Signals PM03
   // Aufruf des Schnittstellen Signal Bausteins / Call the interface signals bool blocks
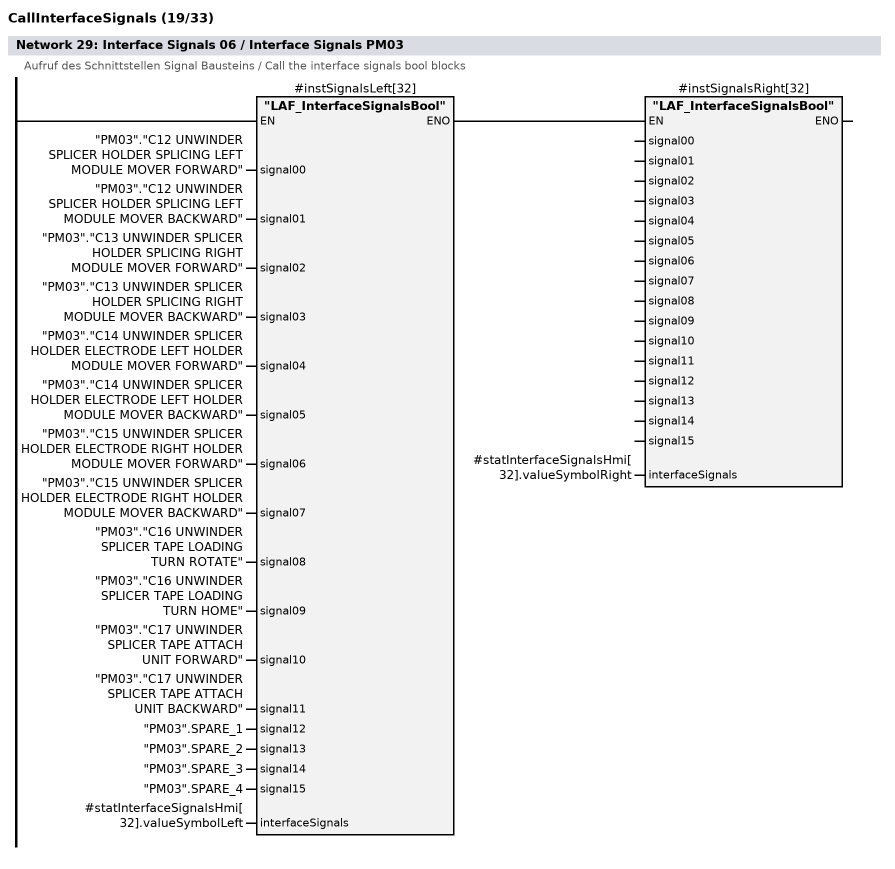
   RUNG wire#powerrail
      #instSignalsLeft[32](signal00 := "PM03"."C12 UNWINDER SPLICER HOLDER SPLICING LEFT MODULE MOVER FORWARD", signal01 := "PM03"."C12 UNWINDER SPLICER HOLDER SPLICING LEFT MODULE MOVER BACKWARD", signal02 := "PM03"."C13 UNWINDER SPLICER HOLDER SPLICING RIGHT MODULE MOVER FORWARD", signal03 := "PM03"."C13 UNWINDER SPLICER HOLDER SPLICING RIGHT MODULE MOVER BACKWARD", signal04 := "PM03"."C14 UNWINDER SPLICER HOLDER ELECTRODE LEFT HOLDER MODULE MOVER FORWARD", signal05 := "PM03"."C14 UNWINDER SPLICER HOLDER ELECTRODE LEFT HOLDER MODULE MOVER BACKWARD", signal06 := "PM03"."C15 UNWINDER SPLICER HOLDER ELECTRODE RIGHT HOLDER MODULE MOVER FORWARD", signal07 := "PM03"."C15 UNWINDER SPLICER HOLDER ELECTRODE RIGHT HOLDER MODULE MOVER BACKWARD", signal08 := "PM03"."C16 UNWINDER SPLICER TAPE LOADING TURN ROTATE", signal09 := "PM03"."C16 UNWINDER SPLICER TAPE LOADING TURN HOME", signal10 := "PM03"."C17 UNWINDER SPLICER TAPE ATTACH UNIT FORWARD", signal11 := "PM03"."C17 UNWINDER SPLICER TAPE ATTACH UNIT BACKWARD", signal12 := "PM03".SPARE_1, signal13 := "PM03".SPARE_2, signal14 := "PM03".SPARE_3, signal15 := "PM03".SPARE_4, interfaceSignals := #statInterfaceSignalsHmi[32].valueSymbolLeft)
      #instSignalsRight[32](signal00 :=, signal01 :=, signal02 :=, signal03 :=, signal04 :=, signal05 :=, signal06 :=, signal07 :=, signal08 :=, signal09 :=, signal10 :=, signal11 :=, signal12 :=, signal13 :=, signal14 :=, signal15 :=, interfaceSignals := #statInterfaceSignalsHmi[32].valueSymbolRight)
   END_RUNG
   // the same network as SCL:
   #instSignalsLeft[32](signal00 := "PM03"."C12 UNWINDER SPLICER HOLDER SPLICING LEFT MODULE MOVER FORWARD",   // "LAF_InterfaceSignalsBool"
                        signal01 := "PM03"."C12 UNWINDER SPLICER HOLDER SPLICING LEFT MODULE MOVER BACKWARD",
                        signal02 := "PM03"."C13 UNWINDER SPLICER HOLDER SPLICING RIGHT MODULE MOVER FORWARD",
                        signal03 := "PM03"."C13 UNWINDER SPLICER HOLDER SPLICING RIGHT MODULE MOVER BACKWARD",
                        signal04 := "PM03"."C14 UNWINDER SPLICER HOLDER ELECTRODE LEFT HOLDER MODULE MOVER FORWARD",
                        signal05 := "PM03"."C14 UNWINDER SPLICER HOLDER ELECTRODE LEFT HOLDER MODULE MOVER BACKWARD",
                        signal06 := "PM03"."C15 UNWINDER SPLICER HOLDER ELECTRODE RIGHT HOLDER MODULE MOVER FORWARD",
                        signal07 := "PM03"."C15 UNWINDER SPLICER HOLDER ELECTRODE RIGHT HOLDER MODULE MOVER BACKWARD",
                        signal08 := "PM03"."C16 UNWINDER SPLICER TAPE LOADING TURN ROTATE",
                        signal09 := "PM03"."C16 UNWINDER SPLICER TAPE LOADING TURN HOME",
                        signal10 := "PM03"."C17 UNWINDER SPLICER TAPE ATTACH UNIT FORWARD",
                        signal11 := "PM03"."C17 UNWINDER SPLICER TAPE ATTACH UNIT BACKWARD",
                        signal12 := "PM03".SPARE_1,
                        signal13 := "PM03".SPARE_2,
                        signal14 := "PM03".SPARE_3,
                        signal15 := "PM03".SPARE_4,
                        interfaceSignals := #statInterfaceSignalsHmi[32].valueSymbolLeft,
                        ENO => #_w1);
   IF #_w1 THEN
       #instSignalsRight[32](interfaceSignals := #statInterfaceSignalsHmi[32].valueSymbolRight);   // "LAF_InterfaceSignalsBool"
   END_IF;
END_REGION

REGION Network 30: Interface Signals 06 / Interface Signals PM04
   // Aufruf des Schnittstellen Signal Bausteins / Call the interface signals bool blocks
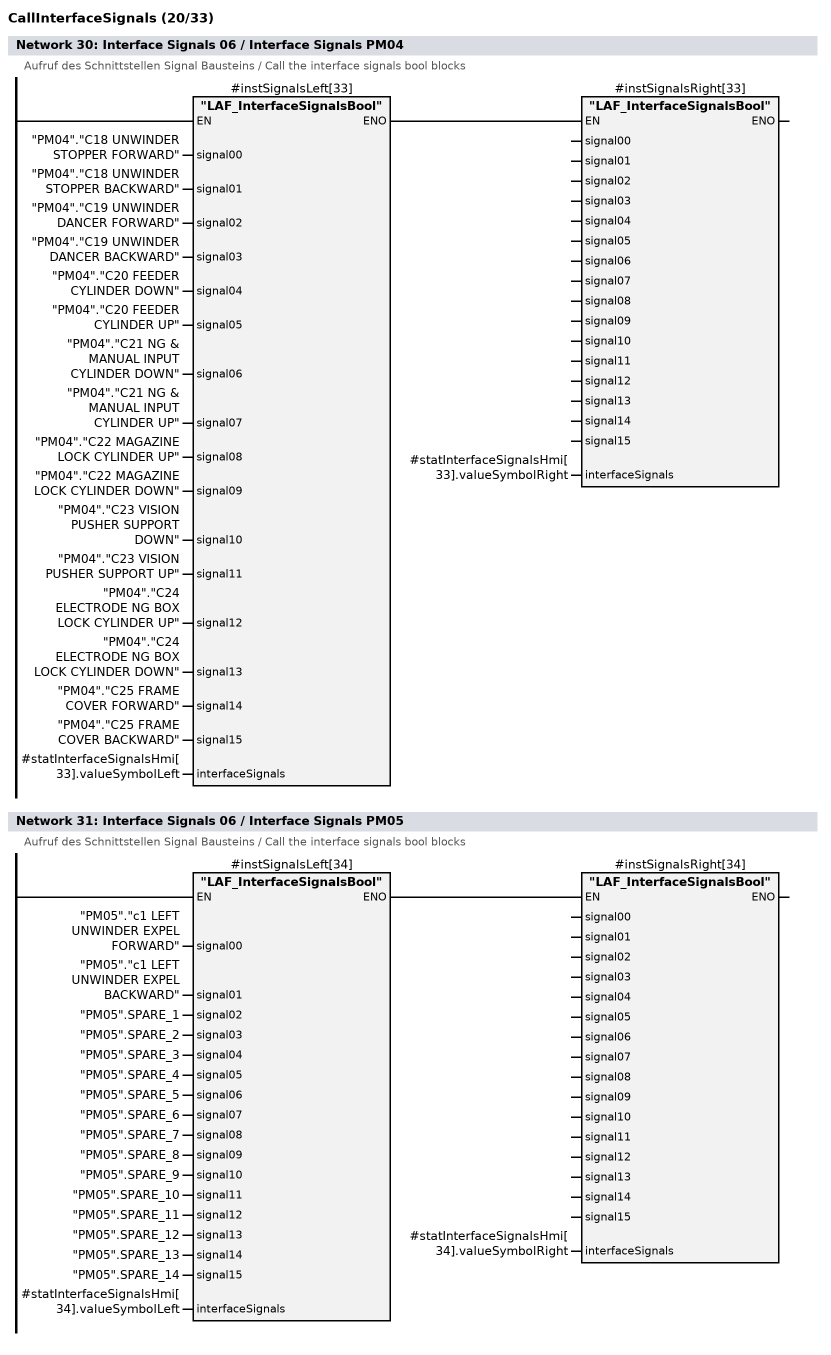
   RUNG wire#powerrail
      #instSignalsLeft[33](signal00 := "PM04"."C18 UNWINDER STOPPER FORWARD", signal01 := "PM04"."C18 UNWINDER STOPPER BACKWARD", signal02 := "PM04"."C19 UNWINDER DANCER FORWARD", signal03 := "PM04"."C19 UNWINDER DANCER BACKWARD", signal04 := "PM04"."C20 FEEDER CYLINDER DOWN", signal05 := "PM04"."C20 FEEDER CYLINDER UP", signal06 := "PM04"."C21 NG & MANUAL INPUT CYLINDER DOWN", signal07 := "PM04"."C21 NG & MANUAL INPUT CYLINDER UP", signal08 := "PM04"."C22 MAGAZINE LOCK CYLINDER UP", signal09 := "PM04"."C22 MAGAZINE LOCK CYLINDER DOWN", signal10 := "PM04"."C23 VISION PUSHER SUPPORT DOWN", signal11 := "PM04"."C23 VISION PUSHER SUPPORT UP", signal12 := "PM04"."C24 ELECTRODE NG BOX LOCK CYLINDER UP", signal13 := "PM04"."C24 ELECTRODE NG BOX LOCK CYLINDER DOWN", signal14 := "PM04"."C25 FRAME COVER FORWARD", signal15 := "PM04"."C25 FRAME COVER BACKWARD", interfaceSignals := #statInterfaceSignalsHmi[33].valueSymbolLeft)
      #instSignalsRight[33](signal00 :=, signal01 :=, signal02 :=, signal03 :=, signal04 :=, signal05 :=, signal06 :=, signal07 :=, signal08 :=, signal09 :=, signal10 :=, signal11 :=, signal12 :=, signal13 :=, signal14 :=, signal15 :=, interfaceSignals := #statInterfaceSignalsHmi[33].valueSymbolRight)
   END_RUNG
   // the same network as SCL:
   #instSignalsLeft[33](signal00 := "PM04"."C18 UNWINDER STOPPER FORWARD",   // "LAF_InterfaceSignalsBool"
                        signal01 := "PM04"."C18 UNWINDER STOPPER BACKWARD",
                        signal02 := "PM04"."C19 UNWINDER DANCER FORWARD",
                        signal03 := "PM04"."C19 UNWINDER DANCER BACKWARD",
                        signal04 := "PM04"."C20 FEEDER CYLINDER DOWN",
                        signal05 := "PM04"."C20 FEEDER CYLINDER UP",
                        signal06 := "PM04"."C21 NG & MANUAL INPUT CYLINDER DOWN",
                        signal07 := "PM04"."C21 NG & MANUAL INPUT CYLINDER UP",
                        signal08 := "PM04"."C22 MAGAZINE LOCK CYLINDER UP",
                        signal09 := "PM04"."C22 MAGAZINE LOCK CYLINDER DOWN",
                        signal10 := "PM04"."C23 VISION PUSHER SUPPORT DOWN",
                        signal11 := "PM04"."C23 VISION PUSHER SUPPORT UP",
                        signal12 := "PM04"."C24 ELECTRODE NG BOX LOCK CYLINDER UP",
                        signal13 := "PM04"."C24 ELECTRODE NG BOX LOCK CYLINDER DOWN",
                        signal14 := "PM04"."C25 FRAME COVER FORWARD",
                        signal15 := "PM04"."C25 FRAME COVER BACKWARD",
                        interfaceSignals := #statInterfaceSignalsHmi[33].valueSymbolLeft,
                        ENO => #_w1);
   IF #_w1 THEN
       #instSignalsRight[33](interfaceSignals := #statInterfaceSignalsHmi[33].valueSymbolRight);   // "LAF_InterfaceSignalsBool"
   END_IF;
END_REGION

REGION Network 31: Interface Signals 06 / Interface Signals PM05
   // Aufruf des Schnittstellen Signal Bausteins / Call the interface signals bool blocks
   RUNG wire#powerrail
      #instSignalsLeft[34](signal00 := "PM05"."c1 LEFT UNWINDER EXPEL FORWARD", signal01 := "PM05"."c1 LEFT UNWINDER EXPEL BACKWARD", signal02 := "PM05".SPARE_1, signal03 := "PM05".SPARE_2, signal04 := "PM05".SPARE_3, signal05 := "PM05".SPARE_4, signal06 := "PM05".SPARE_5, signal07 := "PM05".SPARE_6, signal08 := "PM05".SPARE_7, signal09 := "PM05".SPARE_8, signal10 := "PM05".SPARE_9, signal11 := "PM05".SPARE_10, signal12 := "PM05".SPARE_11, signal13 := "PM05".SPARE_12, signal14 := "PM05".SPARE_13, signal15 := "PM05".SPARE_14, interfaceSignals := #statInterfaceSignalsHmi[34].valueSymbolLeft)
      #instSignalsRight[34](signal00 :=, signal01 :=, signal02 :=, signal03 :=, signal04 :=, signal05 :=, signal06 :=, signal07 :=, signal08 :=, signal09 :=, signal10 :=, signal11 :=, signal12 :=, signal13 :=, signal14 :=, signal15 :=, interfaceSignals := #statInterfaceSignalsHmi[34].valueSymbolRight)
   END_RUNG
   // the same network as SCL:
   #instSignalsLeft[34](signal00 := "PM05"."c1 LEFT UNWINDER EXPEL FORWARD",   // "LAF_InterfaceSignalsBool"
                        signal01 := "PM05"."c1 LEFT UNWINDER EXPEL BACKWARD",
                        signal02 := "PM05".SPARE_1,
                        signal03 := "PM05".SPARE_2,
                        signal04 := "PM05".SPARE_3,
                        signal05 := "PM05".SPARE_4,
                        signal06 := "PM05".SPARE_5,
                        signal07 := "PM05".SPARE_6,
                        signal08 := "PM05".SPARE_7,
                        signal09 := "PM05".SPARE_8,
                        signal10 := "PM05".SPARE_9,
                        signal11 := "PM05".SPARE_10,
                        signal12 := "PM05".SPARE_11,
                        signal13 := "PM05".SPARE_12,
                        signal14 := "PM05".SPARE_13,
                        signal15 := "PM05".SPARE_14,
                        interfaceSignals := #statInterfaceSignalsHmi[34].valueSymbolLeft,
                        ENO => #_w1);
   IF #_w1 THEN
       #instSignalsRight[34](interfaceSignals := #statInterfaceSignalsHmi[34].valueSymbolRight);   // "LAF_InterfaceSignalsBool"
   END_IF;
END_REGION

REGION Network 32: Interface Signals 06 / Interface Signals PM06
   // Aufruf des Schnittstellen Signal Bausteins / Call the interface signals bool blocks
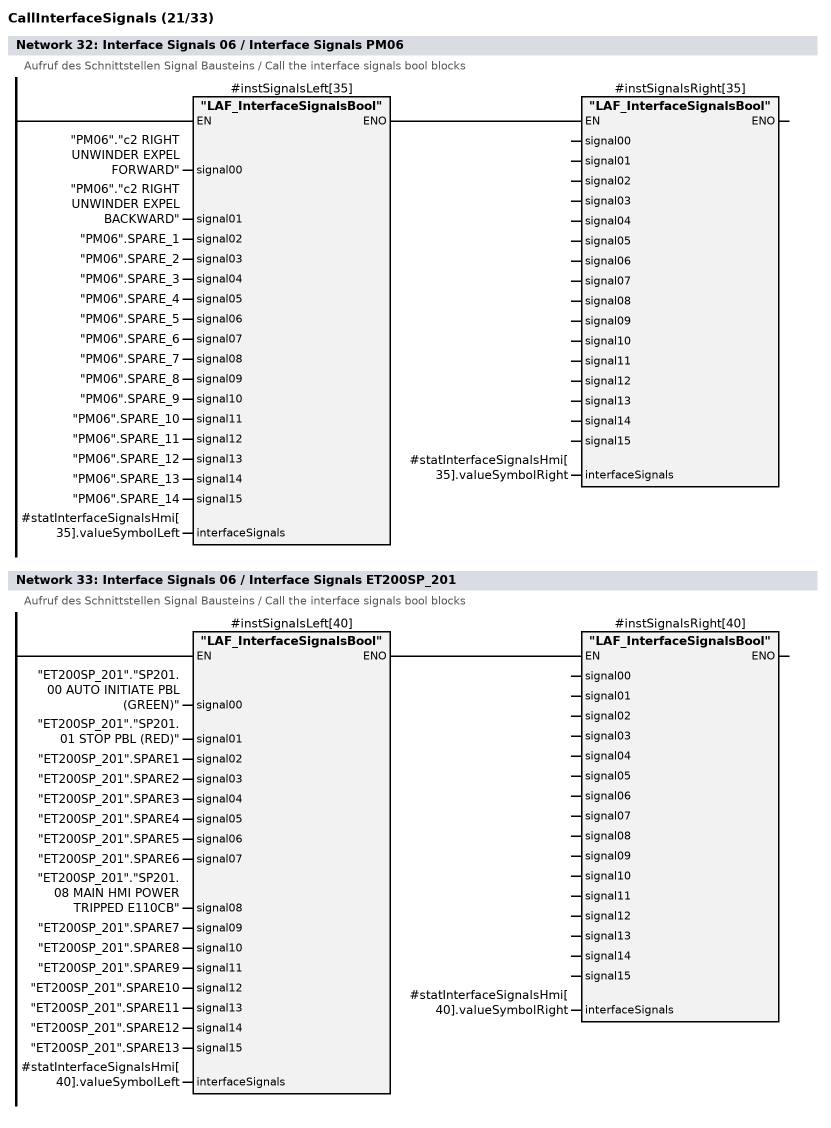
   RUNG wire#powerrail
      #instSignalsLeft[35](signal00 := "PM06"."c2 RIGHT UNWINDER EXPEL FORWARD", signal01 := "PM06"."c2 RIGHT UNWINDER EXPEL BACKWARD", signal02 := "PM06".SPARE_1, signal03 := "PM06".SPARE_2, signal04 := "PM06".SPARE_3, signal05 := "PM06".SPARE_4, signal06 := "PM06".SPARE_5, signal07 := "PM06".SPARE_6, signal08 := "PM06".SPARE_7, signal09 := "PM06".SPARE_8, signal10 := "PM06".SPARE_9, signal11 := "PM06".SPARE_10, signal12 := "PM06".SPARE_11, signal13 := "PM06".SPARE_12, signal14 := "PM06".SPARE_13, signal15 := "PM06".SPARE_14, interfaceSignals := #statInterfaceSignalsHmi[35].valueSymbolLeft)
      #instSignalsRight[35](signal00 :=, signal01 :=, signal02 :=, signal03 :=, signal04 :=, signal05 :=, signal06 :=, signal07 :=, signal08 :=, signal09 :=, signal10 :=, signal11 :=, signal12 :=, signal13 :=, signal14 :=, signal15 :=, interfaceSignals := #statInterfaceSignalsHmi[35].valueSymbolRight)
   END_RUNG
   // the same network as SCL:
   #instSignalsLeft[35](signal00 := "PM06"."c2 RIGHT UNWINDER EXPEL FORWARD",   // "LAF_InterfaceSignalsBool"
                        signal01 := "PM06"."c2 RIGHT UNWINDER EXPEL BACKWARD",
                        signal02 := "PM06".SPARE_1,
                        signal03 := "PM06".SPARE_2,
                        signal04 := "PM06".SPARE_3,
                        signal05 := "PM06".SPARE_4,
                        signal06 := "PM06".SPARE_5,
                        signal07 := "PM06".SPARE_6,
                        signal08 := "PM06".SPARE_7,
                        signal09 := "PM06".SPARE_8,
                        signal10 := "PM06".SPARE_9,
                        signal11 := "PM06".SPARE_10,
                        signal12 := "PM06".SPARE_11,
                        signal13 := "PM06".SPARE_12,
                        signal14 := "PM06".SPARE_13,
                        signal15 := "PM06".SPARE_14,
                        interfaceSignals := #statInterfaceSignalsHmi[35].valueSymbolLeft,
                        ENO => #_w1);
   IF #_w1 THEN
       #instSignalsRight[35](interfaceSignals := #statInterfaceSignalsHmi[35].valueSymbolRight);   // "LAF_InterfaceSignalsBool"
   END_IF;
END_REGION

REGION Network 33: Interface Signals 06 / Interface Signals ET200SP_201
   // Aufruf des Schnittstellen Signal Bausteins / Call the interface signals bool blocks
   RUNG wire#powerrail
      #instSignalsLeft[40](signal00 := "ET200SP_201"."SP201.00 AUTO INITIATE PBL (GREEN)", signal01 := "ET200SP_201"."SP201.01 STOP PBL (RED)", signal02 := "ET200SP_201".SPARE1, signal03 := "ET200SP_201".SPARE2, signal04 := "ET200SP_201".SPARE3, signal05 := "ET200SP_201".SPARE4, signal06 := "ET200SP_201".SPARE5, signal07 := "ET200SP_201".SPARE6, signal08 := "ET200SP_201"."SP201.08 MAIN HMI POWER TRIPPED E110CB", signal09 := "ET200SP_201".SPARE7, signal10 := "ET200SP_201".SPARE8, signal11 := "ET200SP_201".SPARE9, signal12 := "ET200SP_201".SPARE10, signal13 := "ET200SP_201".SPARE11, signal14 := "ET200SP_201".SPARE12, signal15 := "ET200SP_201".SPARE13, interfaceSignals := #statInterfaceSignalsHmi[40].valueSymbolLeft)
      #instSignalsRight[40](signal00 :=, signal01 :=, signal02 :=, signal03 :=, signal04 :=, signal05 :=, signal06 :=, signal07 :=, signal08 :=, signal09 :=, signal10 :=, signal11 :=, signal12 :=, signal13 :=, signal14 :=, signal15 :=, interfaceSignals := #statInterfaceSignalsHmi[40].valueSymbolRight)
   END_RUNG
   // the same network as SCL:
   #instSignalsLeft[40](signal00 := "ET200SP_201"."SP201.00 AUTO INITIATE PBL (GREEN)",   // "LAF_InterfaceSignalsBool"
                        signal01 := "ET200SP_201"."SP201.01 STOP PBL (RED)",
                        signal02 := "ET200SP_201".SPARE1,
                        signal03 := "ET200SP_201".SPARE2,
                        signal04 := "ET200SP_201".SPARE3,
                        signal05 := "ET200SP_201".SPARE4,
                        signal06 := "ET200SP_201".SPARE5,
                        signal07 := "ET200SP_201".SPARE6,
                        signal08 := "ET200SP_201"."SP201.08 MAIN HMI POWER TRIPPED E110CB",
                        signal09 := "ET200SP_201".SPARE7,
                        signal10 := "ET200SP_201".SPARE8,
                        signal11 := "ET200SP_201".SPARE9,
                        signal12 := "ET200SP_201".SPARE10,
                        signal13 := "ET200SP_201".SPARE11,
                        signal14 := "ET200SP_201".SPARE12,
                        signal15 := "ET200SP_201".SPARE13,
                        interfaceSignals := #statInterfaceSignalsHmi[40].valueSymbolLeft,
                        ENO => #_w1);
   IF #_w1 THEN
       #instSignalsRight[40](interfaceSignals := #statInterfaceSignalsHmi[40].valueSymbolRight);   // "LAF_InterfaceSignalsBool"
   END_IF;
END_REGION

REGION Network 34: Interface Signals 06 / Interface Signals ET200SP_202
   // Aufruf des Schnittstellen Signal Bausteins / Call the interface signals bool blocks
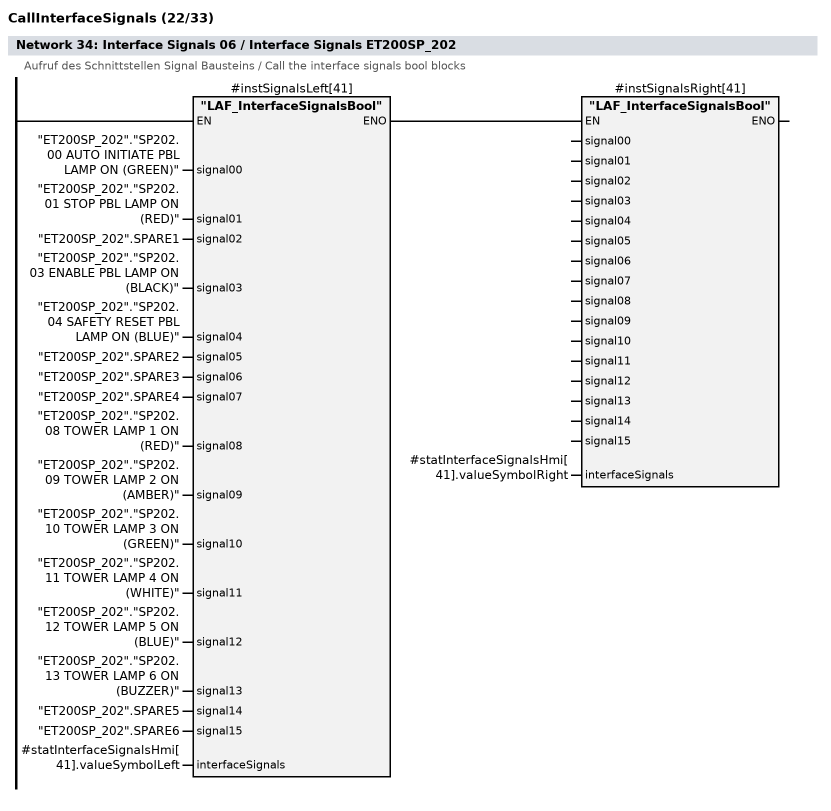
   RUNG wire#powerrail
      #instSignalsLeft[41](signal00 := "ET200SP_202"."SP202.00 AUTO INITIATE PBL LAMP ON (GREEN)", signal01 := "ET200SP_202"."SP202.01 STOP PBL LAMP ON (RED)", signal02 := "ET200SP_202".SPARE1, signal03 := "ET200SP_202"."SP202.03 ENABLE PBL LAMP ON (BLACK)", signal04 := "ET200SP_202"."SP202.04 SAFETY RESET PBL LAMP ON (BLUE)", signal05 := "ET200SP_202".SPARE2, signal06 := "ET200SP_202".SPARE3, signal07 := "ET200SP_202".SPARE4, signal08 := "ET200SP_202"."SP202.08 TOWER LAMP 1 ON (RED)", signal09 := "ET200SP_202"."SP202.09 TOWER LAMP 2 ON (AMBER)", signal10 := "ET200SP_202"."SP202.10 TOWER LAMP 3 ON (GREEN)", signal11 := "ET200SP_202"."SP202.11 TOWER LAMP 4 ON (WHITE)", signal12 := "ET200SP_202"."SP202.12 TOWER LAMP 5 ON (BLUE)", signal13 := "ET200SP_202"."SP202.13 TOWER LAMP 6 ON (BUZZER)", signal14 := "ET200SP_202".SPARE5, signal15 := "ET200SP_202".SPARE6, interfaceSignals := #statInterfaceSignalsHmi[41].valueSymbolLeft)
      #instSignalsRight[41](signal00 :=, signal01 :=, signal02 :=, signal03 :=, signal04 :=, signal05 :=, signal06 :=, signal07 :=, signal08 :=, signal09 :=, signal10 :=, signal11 :=, signal12 :=, signal13 :=, signal14 :=, signal15 :=, interfaceSignals := #statInterfaceSignalsHmi[41].valueSymbolRight)
   END_RUNG
   // the same network as SCL:
   #instSignalsLeft[41](signal00 := "ET200SP_202"."SP202.00 AUTO INITIATE PBL LAMP ON (GREEN)",   // "LAF_InterfaceSignalsBool"
                        signal01 := "ET200SP_202"."SP202.01 STOP PBL LAMP ON (RED)",
                        signal02 := "ET200SP_202".SPARE1,
                        signal03 := "ET200SP_202"."SP202.03 ENABLE PBL LAMP ON (BLACK)",
                        signal04 := "ET200SP_202"."SP202.04 SAFETY RESET PBL LAMP ON (BLUE)",
                        signal05 := "ET200SP_202".SPARE2,
                        signal06 := "ET200SP_202".SPARE3,
                        signal07 := "ET200SP_202".SPARE4,
                        signal08 := "ET200SP_202"."SP202.08 TOWER LAMP 1 ON (RED)",
                        signal09 := "ET200SP_202"."SP202.09 TOWER LAMP 2 ON (AMBER)",
                        signal10 := "ET200SP_202"."SP202.10 TOWER LAMP 3 ON (GREEN)",
                        signal11 := "ET200SP_202"."SP202.11 TOWER LAMP 4 ON (WHITE)",
                        signal12 := "ET200SP_202"."SP202.12 TOWER LAMP 5 ON (BLUE)",
                        signal13 := "ET200SP_202"."SP202.13 TOWER LAMP 6 ON (BUZZER)",
                        signal14 := "ET200SP_202".SPARE5,
                        signal15 := "ET200SP_202".SPARE6,
                        interfaceSignals := #statInterfaceSignalsHmi[41].valueSymbolLeft,
                        ENO => #_w1);
   IF #_w1 THEN
       #instSignalsRight[41](interfaceSignals := #statInterfaceSignalsHmi[41].valueSymbolRight);   // "LAF_InterfaceSignalsBool"
   END_IF;
END_REGION

REGION Network 35: Interface Signals 06 / Interface Signals ET200SP_203
   // Aufruf des Schnittstellen Signal Bausteins / Call the interface signals bool blocks
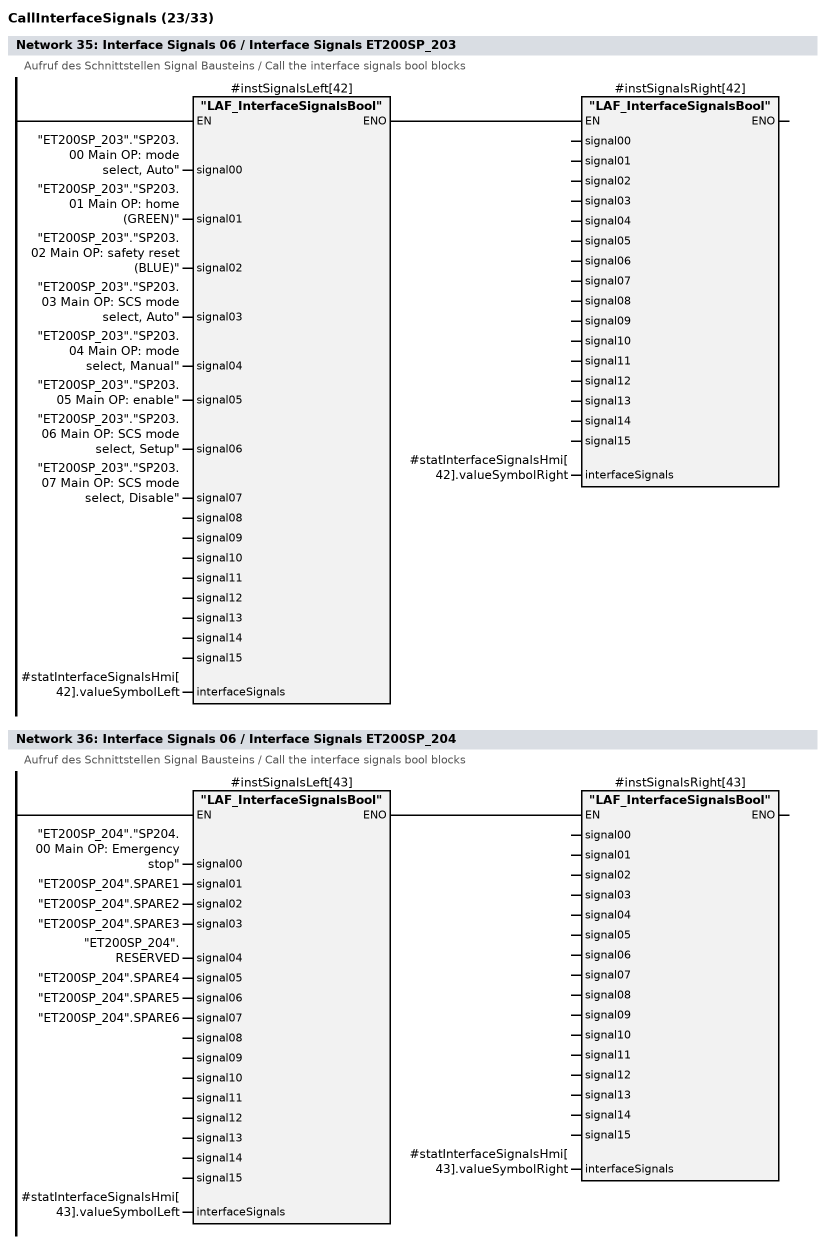
   RUNG wire#powerrail
      #instSignalsLeft[42](signal00 := "ET200SP_203"."SP203.00 Main OP: mode select, Auto", signal01 := "ET200SP_203"."SP203.01 Main OP: home (GREEN)", signal02 := "ET200SP_203"."SP203.02 Main OP: safety reset (BLUE)", signal03 := "ET200SP_203"."SP203.03 Main OP: SCS mode select, Auto", signal04 := "ET200SP_203"."SP203.04 Main OP: mode select, Manual", signal05 := "ET200SP_203"."SP203.05 Main OP: enable", signal06 := "ET200SP_203"."SP203.06 Main OP: SCS mode select, Setup", signal07 := "ET200SP_203"."SP203.07 Main OP: SCS mode select, Disable", signal08 :=, signal09 :=, signal10 :=, signal11 :=, signal12 :=, signal13 :=, signal14 :=, signal15 :=, interfaceSignals := #statInterfaceSignalsHmi[42].valueSymbolLeft)
      #instSignalsRight[42](signal00 :=, signal01 :=, signal02 :=, signal03 :=, signal04 :=, signal05 :=, signal06 :=, signal07 :=, signal08 :=, signal09 :=, signal10 :=, signal11 :=, signal12 :=, signal13 :=, signal14 :=, signal15 :=, interfaceSignals := #statInterfaceSignalsHmi[42].valueSymbolRight)
   END_RUNG
   // the same network as SCL:
   #instSignalsLeft[42](signal00 := "ET200SP_203"."SP203.00 Main OP: mode select, Auto",   // "LAF_InterfaceSignalsBool"
                        signal01 := "ET200SP_203"."SP203.01 Main OP: home (GREEN)",
                        signal02 := "ET200SP_203"."SP203.02 Main OP: safety reset (BLUE)",
                        signal03 := "ET200SP_203"."SP203.03 Main OP: SCS mode select, Auto",
                        signal04 := "ET200SP_203"."SP203.04 Main OP: mode select, Manual",
                        signal05 := "ET200SP_203"."SP203.05 Main OP: enable",
                        signal06 := "ET200SP_203"."SP203.06 Main OP: SCS mode select, Setup",
                        signal07 := "ET200SP_203"."SP203.07 Main OP: SCS mode select, Disable",
                        interfaceSignals := #statInterfaceSignalsHmi[42].valueSymbolLeft,
                        ENO => #_w1);
   IF #_w1 THEN
       #instSignalsRight[42](interfaceSignals := #statInterfaceSignalsHmi[42].valueSymbolRight);   // "LAF_InterfaceSignalsBool"
   END_IF;
END_REGION

